(* Logix 5000 project; controller TBEN_Lx_8IOL_AOI_V0_2 vendor 1 type 14 code 176 rev 32.11; software revision 32.00; part 12 of 16 *)

           TBEN_L4_8IOL1:O.Data[69].10   // IO-Link Port 5 - Output data word 3 (INT bit10)
           TBEN_L4_8IOL1:O.Data[69].11   // IO-Link Port 5 - Output data word 3 (INT bit11)
           TBEN_L4_8IOL1:O.Data[69].12   // IO-Link Port 5 - Output data word 3 (INT bit12)
           TBEN_L4_8IOL1:O.Data[69].13   // IO-Link Port 5 - Output data word 3 (INT bit13)
           TBEN_L4_8IOL1:O.Data[69].14   // IO-Link Port 5 - Output data word 3 (INT bit14)
           TBEN_L4_8IOL1:O.Data[69].15   // IO-Link Port 5 - Output data word 3 (INT bit15)
           TBEN_L4_8IOL1:O.Data[69].2   // IO-Link Port 5 - Output data word 3 (INT bit2)
           TBEN_L4_8IOL1:O.Data[69].3   // IO-Link Port 5 - Output data word 3 (INT bit3)
           TBEN_L4_8IOL1:O.Data[69].4   // IO-Link Port 5 - Output data word 3 (INT bit4)
           TBEN_L4_8IOL1:O.Data[69].5   // IO-Link Port 5 - Output data word 3 (INT bit5)
           TBEN_L4_8IOL1:O.Data[69].6   // IO-Link Port 5 - Output data word 3 (INT bit6)
           TBEN_L4_8IOL1:O.Data[69].7   // IO-Link Port 5 - Output data word 3 (INT bit7)
           TBEN_L4_8IOL1:O.Data[69].8   // IO-Link Port 5 - Output data word 3 (INT bit8)
           TBEN_L4_8IOL1:O.Data[69].9   // IO-Link Port 5 - Output data word 3 (INT bit9)
           TBEN_L4_8IOL1:O.Data[6]   // IO-Link Port 1 - Output data word 4
           TBEN_L4_8IOL1:O.Data[6].0   // IO-Link Port 1 - Output data word 4 (INT bit0)
           TBEN_L4_8IOL1:O.Data[6].1   // IO-Link Port 1 - Output data word 4 (INT bit1)
           TBEN_L4_8IOL1:O.Data[6].10   // IO-Link Port 1 - Output data word 4 (INT bit10)
           TBEN_L4_8IOL1:O.Data[6].11   // IO-Link Port 1 - Output data word 4 (INT bit11)
           TBEN_L4_8IOL1:O.Data[6].12   // IO-Link Port 1 - Output data word 4 (INT bit12)
           TBEN_L4_8IOL1:O.Data[6].13   // IO-Link Port 1 - Output data word 4 (INT bit13)
           TBEN_L4_8IOL1:O.Data[6].14   // IO-Link Port 1 - Output data word 4 (INT bit14)
           TBEN_L4_8IOL1:O.Data[6].15   // IO-Link Port 1 - Output data word 4 (INT bit15)
           TBEN_L4_8IOL1:O.Data[6].2   // IO-Link Port 1 - Output data word 4 (INT bit2)
           TBEN_L4_8IOL1:O.Data[6].3   // IO-Link Port 1 - Output data word 4 (INT bit3)
           TBEN_L4_8IOL1:O.Data[6].4   // IO-Link Port 1 - Output data word 4 (INT bit4)
           TBEN_L4_8IOL1:O.Data[6].5   // IO-Link Port 1 - Output data word 4 (INT bit5)
           TBEN_L4_8IOL1:O.Data[6].6   // IO-Link Port 1 - Output data word 4 (INT bit6)
           TBEN_L4_8IOL1:O.Data[6].7   // IO-Link Port 1 - Output data word 4 (INT bit7)
           TBEN_L4_8IOL1:O.Data[6].8   // IO-Link Port 1 - Output data word 4 (INT bit8)
           TBEN_L4_8IOL1:O.Data[6].9   // IO-Link Port 1 - Output data word 4 (INT bit9)
           TBEN_L4_8IOL1:O.Data[70]   // IO-Link Port 5 - Output data word 4
           TBEN_L4_8IOL1:O.Data[70].0   // IO-Link Port 5 - Output data word 4 (INT bit0)
           TBEN_L4_8IOL1:O.Data[70].1   // IO-Link Port 5 - Output data word 4 (INT bit1)
           TBEN_L4_8IOL1:O.Data[70].10   // IO-Link Port 5 - Output data word 4 (INT bit10)
           TBEN_L4_8IOL1:O.Data[70].11   // IO-Link Port 5 - Output data word 4 (INT bit11)
           TBEN_L4_8IOL1:O.Data[70].12   // IO-Link Port 5 - Output data word 4 (INT bit12)
           TBEN_L4_8IOL1:O.Data[70].13   // IO-Link Port 5 - Output data word 4 (INT bit13)
           TBEN_L4_8IOL1:O.Data[70].14   // IO-Link Port 5 - Output data word 4 (INT bit14)
           TBEN_L4_8IOL1:O.Data[70].15   // IO-Link Port 5 - Output data word 4 (INT bit15)
           TBEN_L4_8IOL1:O.Data[70].2   // IO-Link Port 5 - Output data word 4 (INT bit2)
           TBEN_L4_8IOL1:O.Data[70].3   // IO-Link Port 5 - Output data word 4 (INT bit3)
           TBEN_L4_8IOL1:O.Data[70].4   // IO-Link Port 5 - Output data word 4 (INT bit4)
           TBEN_L4_8IOL1:O.Data[70].5   // IO-Link Port 5 - Output data word 4 (INT bit5)
           TBEN_L4_8IOL1:O.Data[70].6   // IO-Link Port 5 - Output data word 4 (INT bit6)
           TBEN_L4_8IOL1:O.Data[70].7   // IO-Link Port 5 - Output data word 4 (INT bit7)
           TBEN_L4_8IOL1:O.Data[70].8   // IO-Link Port 5 - Output data word 4 (INT bit8)
           TBEN_L4_8IOL1:O.Data[70].9   // IO-Link Port 5 - Output data word 4 (INT bit9)
           TBEN_L4_8IOL1:O.Data[71]   // IO-Link Port 5 - Output data word 5
           TBEN_L4_8IOL1:O.Data[71].0   // IO-Link Port 5 - Output data word 5 (INT bit0)
           TBEN_L4_8IOL1:O.Data[71].1   // IO-Link Port 5 - Output data word 5 (INT bit1)
           TBEN_L4_8IOL1:O.Data[71].10   // IO-Link Port 5 - Output data word 5 (INT bit10)
           TBEN_L4_8IOL1:O.Data[71].11   // IO-Link Port 5 - Output data word 5 (INT bit11)
           TBEN_L4_8IOL1:O.Data[71].12   // IO-Link Port 5 - Output data word 5 (INT bit12)
           TBEN_L4_8IOL1:O.Data[71].13   // IO-Link Port 5 - Output data word 5 (INT bit13)
           TBEN_L4_8IOL1:O.Data[71].14   // IO-Link Port 5 - Output data word 5 (INT bit14)
           TBEN_L4_8IOL1:O.Data[71].15   // IO-Link Port 5 - Output data word 5 (INT bit15)
           TBEN_L4_8IOL1:O.Data[71].2   // IO-Link Port 5 - Output data word 5 (INT bit2)
           TBEN_L4_8IOL1:O.Data[71].3   // IO-Link Port 5 - Output data word 5 (INT bit3)
           TBEN_L4_8IOL1:O.Data[71].4   // IO-Link Port 5 - Output data word 5 (INT bit4)
           TBEN_L4_8IOL1:O.Data[71].5   // IO-Link Port 5 - Output data word 5 (INT bit5)
           TBEN_L4_8IOL1:O.Data[71].6   // IO-Link Port 5 - Output data word 5 (INT bit6)
           TBEN_L4_8IOL1:O.Data[71].7   // IO-Link Port 5 - Output data word 5 (INT bit7)
           TBEN_L4_8IOL1:O.Data[71].8   // IO-Link Port 5 - Output data word 5 (INT bit8)
           TBEN_L4_8IOL1:O.Data[71].9   // IO-Link Port 5 - Output data word 5 (INT bit9)
           TBEN_L4_8IOL1:O.Data[72]   // IO-Link Port 5 - Output data word 6
           TBEN_L4_8IOL1:O.Data[72].0   // IO-Link Port 5 - Output data word 6 (INT bit0)
           TBEN_L4_8IOL1:O.Data[72].1   // IO-Link Port 5 - Output data word 6 (INT bit1)
           TBEN_L4_8IOL1:O.Data[72].10   // IO-Link Port 5 - Output data word 6 (INT bit10)
           TBEN_L4_8IOL1:O.Data[72].11   // IO-Link Port 5 - Output data word 6 (INT bit11)
           TBEN_L4_8IOL1:O.Data[72].12   // IO-Link Port 5 - Output data word 6 (INT bit12)
           TBEN_L4_8IOL1:O.Data[72].13   // IO-Link Port 5 - Output data word 6 (INT bit13)
           TBEN_L4_8IOL1:O.Data[72].14   // IO-Link Port 5 - Output data word 6 (INT bit14)
           TBEN_L4_8IOL1:O.Data[72].15   // IO-Link Port 5 - Output data word 6 (INT bit15)
           TBEN_L4_8IOL1:O.Data[72].2   // IO-Link Port 5 - Output data word 6 (INT bit2)
           TBEN_L4_8IOL1:O.Data[72].3   // IO-Link Port 5 - Output data word 6 (INT bit3)
           TBEN_L4_8IOL1:O.Data[72].4   // IO-Link Port 5 - Output data word 6 (INT bit4)
           TBEN_L4_8IOL1:O.Data[72].5   // IO-Link Port 5 - Output data word 6 (INT bit5)
           TBEN_L4_8IOL1:O.Data[72].6   // IO-Link Port 5 - Output data word 6 (INT bit6)
           TBEN_L4_8IOL1:O.Data[72].7   // IO-Link Port 5 - Output data word 6 (INT bit7)
           TBEN_L4_8IOL1:O.Data[72].8   // IO-Link Port 5 - Output data word 6 (INT bit8)
           TBEN_L4_8IOL1:O.Data[72].9   // IO-Link Port 5 - Output data word 6 (INT bit9)
           TBEN_L4_8IOL1:O.Data[73]   // IO-Link Port 5 - Output data word 7
           TBEN_L4_8IOL1:O.Data[73].0   // IO-Link Port 5 - Output data word 7 (INT bit0)
           TBEN_L4_8IOL1:O.Data[73].1   // IO-Link Port 5 - Output data word 7 (INT bit1)
           TBEN_L4_8IOL1:O.Data[73].10   // IO-Link Port 5 - Output data word 7 (INT bit10)
           TBEN_L4_8IOL1:O.Data[73].11   // IO-Link Port 5 - Output data word 7 (INT bit11)
           TBEN_L4_8IOL1:O.Data[73].12   // IO-Link Port 5 - Output data word 7 (INT bit12)
           TBEN_L4_8IOL1:O.Data[73].13   // IO-Link Port 5 - Output data word 7 (INT bit13)
           TBEN_L4_8IOL1:O.Data[73].14   // IO-Link Port 5 - Output data word 7 (INT bit14)
           TBEN_L4_8IOL1:O.Data[73].15   // IO-Link Port 5 - Output data word 7 (INT bit15)
           TBEN_L4_8IOL1:O.Data[73].2   // IO-Link Port 5 - Output data word 7 (INT bit2)
           TBEN_L4_8IOL1:O.Data[73].3   // IO-Link Port 5 - Output data word 7 (INT bit3)
           TBEN_L4_8IOL1:O.Data[73].4   // IO-Link Port 5 - Output data word 7 (INT bit4)
           TBEN_L4_8IOL1:O.Data[73].5   // IO-Link Port 5 - Output data word 7 (INT bit5)
           TBEN_L4_8IOL1:O.Data[73].6   // IO-Link Port 5 - Output data word 7 (INT bit6)
           TBEN_L4_8IOL1:O.Data[73].7   // IO-Link Port 5 - Output data word 7 (INT bit7)
           TBEN_L4_8IOL1:O.Data[73].8   // IO-Link Port 5 - Output data word 7 (INT bit8)
           TBEN_L4_8IOL1:O.Data[73].9   // IO-Link Port 5 - Output data word 7 (INT bit9)
           TBEN_L4_8IOL1:O.Data[74]   // IO-Link Port 5 - Output data word 8
           TBEN_L4_8IOL1:O.Data[74].0   // IO-Link Port 5 - Output data word 8 (INT bit0)
           TBEN_L4_8IOL1:O.Data[74].1   // IO-Link Port 5 - Output data word 8 (INT bit1)
           TBEN_L4_8IOL1:O.Data[74].10   // IO-Link Port 5 - Output data word 8 (INT bit10)
           TBEN_L4_8IOL1:O.Data[74].11   // IO-Link Port 5 - Output data word 8 (INT bit11)
           TBEN_L4_8IOL1:O.Data[74].12   // IO-Link Port 5 - Output data word 8 (INT bit12)
           TBEN_L4_8IOL1:O.Data[74].13   // IO-Link Port 5 - Output data word 8 (INT bit13)
           TBEN_L4_8IOL1:O.Data[74].14   // IO-Link Port 5 - Output data word 8 (INT bit14)
           TBEN_L4_8IOL1:O.Data[74].15   // IO-Link Port 5 - Output data word 8 (INT bit15)
           TBEN_L4_8IOL1:O.Data[74].2   // IO-Link Port 5 - Output data word 8 (INT bit2)
           TBEN_L4_8IOL1:O.Data[74].3   // IO-Link Port 5 - Output data word 8 (INT bit3)
           TBEN_L4_8IOL1:O.Data[74].4   // IO-Link Port 5 - Output data word 8 (INT bit4)
           TBEN_L4_8IOL1:O.Data[74].5   // IO-Link Port 5 - Output data word 8 (INT bit5)
           TBEN_L4_8IOL1:O.Data[74].6   // IO-Link Port 5 - Output data word 8 (INT bit6)
           TBEN_L4_8IOL1:O.Data[74].7   // IO-Link Port 5 - Output data word 8 (INT bit7)
           TBEN_L4_8IOL1:O.Data[74].8   // IO-Link Port 5 - Output data word 8 (INT bit8)
           TBEN_L4_8IOL1:O.Data[74].9   // IO-Link Port 5 - Output data word 8 (INT bit9)
           TBEN_L4_8IOL1:O.Data[75]   // IO-Link Port 5 - Output data word 9
           TBEN_L4_8IOL1:O.Data[75].0   // IO-Link Port 5 - Output data word 9 (INT bit0)
           TBEN_L4_8IOL1:O.Data[75].1   // IO-Link Port 5 - Output data word 9 (INT bit1)
           TBEN_L4_8IOL1:O.Data[75].10   // IO-Link Port 5 - Output data word 9 (INT bit10)
           TBEN_L4_8IOL1:O.Data[75].11   // IO-Link Port 5 - Output data word 9 (INT bit11)
           TBEN_L4_8IOL1:O.Data[75].12   // IO-Link Port 5 - Output data word 9 (INT bit12)
           TBEN_L4_8IOL1:O.Data[75].13   // IO-Link Port 5 - Output data word 9 (INT bit13)
           TBEN_L4_8IOL1:O.Data[75].14   // IO-Link Port 5 - Output data word 9 (INT bit14)
           TBEN_L4_8IOL1:O.Data[75].15   // IO-Link Port 5 - Output data word 9 (INT bit15)
           TBEN_L4_8IOL1:O.Data[75].2   // IO-Link Port 5 - Output data word 9 (INT bit2)
           TBEN_L4_8IOL1:O.Data[75].3   // IO-Link Port 5 - Output data word 9 (INT bit3)
           TBEN_L4_8IOL1:O.Data[75].4   // IO-Link Port 5 - Output data word 9 (INT bit4)
           TBEN_L4_8IOL1:O.Data[75].5   // IO-Link Port 5 - Output data word 9 (INT bit5)
           TBEN_L4_8IOL1:O.Data[75].6   // IO-Link Port 5 - Output data word 9 (INT bit6)
           TBEN_L4_8IOL1:O.Data[75].7   // IO-Link Port 5 - Output data word 9 (INT bit7)
           TBEN_L4_8IOL1:O.Data[75].8   // IO-Link Port 5 - Output data word 9 (INT bit8)
           TBEN_L4_8IOL1:O.Data[75].9   // IO-Link Port 5 - Output data word 9 (INT bit9)
           TBEN_L4_8IOL1:O.Data[76]   // IO-Link Port 5 - Output data word 10
           TBEN_L4_8IOL1:O.Data[76].0   // IO-Link Port 5 - Output data word 10 (INT bit0)
           TBEN_L4_8IOL1:O.Data[76].1   // IO-Link Port 5 - Output data word 10 (INT bit1)
           TBEN_L4_8IOL1:O.Data[76].10   // IO-Link Port 5 - Output data word 10 (INT bit10)
           TBEN_L4_8IOL1:O.Data[76].11   // IO-Link Port 5 - Output data word 10 (INT bit11)
           TBEN_L4_8IOL1:O.Data[76].12   // IO-Link Port 5 - Output data word 10 (INT bit12)
           TBEN_L4_8IOL1:O.Data[76].13   // IO-Link Port 5 - Output data word 10 (INT bit13)
           TBEN_L4_8IOL1:O.Data[76].14   // IO-Link Port 5 - Output data word 10 (INT bit14)
           TBEN_L4_8IOL1:O.Data[76].15   // IO-Link Port 5 - Output data word 10 (INT bit15)
           TBEN_L4_8IOL1:O.Data[76].2   // IO-Link Port 5 - Output data word 10 (INT bit2)
           TBEN_L4_8IOL1:O.Data[76].3   // IO-Link Port 5 - Output data word 10 (INT bit3)
           TBEN_L4_8IOL1:O.Data[76].4   // IO-Link Port 5 - Output data word 10 (INT bit4)
           TBEN_L4_8IOL1:O.Data[76].5   // IO-Link Port 5 - Output data word 10 (INT bit5)
           TBEN_L4_8IOL1:O.Data[76].6   // IO-Link Port 5 - Output data word 10 (INT bit6)
           TBEN_L4_8IOL1:O.Data[76].7   // IO-Link Port 5 - Output data word 10 (INT bit7)
           TBEN_L4_8IOL1:O.Data[76].8   // IO-Link Port 5 - Output data word 10 (INT bit8)
           TBEN_L4_8IOL1:O.Data[76].9   // IO-Link Port 5 - Output data word 10 (INT bit9)
           TBEN_L4_8IOL1:O.Data[77]   // IO-Link Port 5 - Output data word 11
           TBEN_L4_8IOL1:O.Data[77].0   // IO-Link Port 5 - Output data word 11 (INT bit0)
           TBEN_L4_8IOL1:O.Data[77].1   // IO-Link Port 5 - Output data word 11 (INT bit1)
           TBEN_L4_8IOL1:O.Data[77].10   // IO-Link Port 5 - Output data word 11 (INT bit10)
           TBEN_L4_8IOL1:O.Data[77].11   // IO-Link Port 5 - Output data word 11 (INT bit11)
           TBEN_L4_8IOL1:O.Data[77].12   // IO-Link Port 5 - Output data word 11 (INT bit12)
           TBEN_L4_8IOL1:O.Data[77].13   // IO-Link Port 5 - Output data word 11 (INT bit13)
           TBEN_L4_8IOL1:O.Data[77].14   // IO-Link Port 5 - Output data word 11 (INT bit14)
           TBEN_L4_8IOL1:O.Data[77].15   // IO-Link Port 5 - Output data word 11 (INT bit15)
           TBEN_L4_8IOL1:O.Data[77].2   // IO-Link Port 5 - Output data word 11 (INT bit2)
           TBEN_L4_8IOL1:O.Data[77].3   // IO-Link Port 5 - Output data word 11 (INT bit3)
           TBEN_L4_8IOL1:O.Data[77].4   // IO-Link Port 5 - Output data word 11 (INT bit4)
           TBEN_L4_8IOL1:O.Data[77].5   // IO-Link Port 5 - Output data word 11 (INT bit5)
           TBEN_L4_8IOL1:O.Data[77].6   // IO-Link Port 5 - Output data word 11 (INT bit6)
           TBEN_L4_8IOL1:O.Data[77].7   // IO-Link Port 5 - Output data word 11 (INT bit7)
           TBEN_L4_8IOL1:O.Data[77].8   // IO-Link Port 5 - Output data word 11 (INT bit8)
           TBEN_L4_8IOL1:O.Data[77].9   // IO-Link Port 5 - Output data word 11 (INT bit9)
           TBEN_L4_8IOL1:O.Data[78]   // IO-Link Port 5 - Output data word 12
           TBEN_L4_8IOL1:O.Data[78].0   // IO-Link Port 5 - Output data word 12 (INT bit0)
           TBEN_L4_8IOL1:O.Data[78].1   // IO-Link Port 5 - Output data word 12 (INT bit1)
           TBEN_L4_8IOL1:O.Data[78].10   // IO-Link Port 5 - Output data word 12 (INT bit10)
           TBEN_L4_8IOL1:O.Data[78].11   // IO-Link Port 5 - Output data word 12 (INT bit11)
           TBEN_L4_8IOL1:O.Data[78].12   // IO-Link Port 5 - Output data word 12 (INT bit12)
           TBEN_L4_8IOL1:O.Data[78].13   // IO-Link Port 5 - Output data word 12 (INT bit13)
           TBEN_L4_8IOL1:O.Data[78].14   // IO-Link Port 5 - Output data word 12 (INT bit14)
           TBEN_L4_8IOL1:O.Data[78].15   // IO-Link Port 5 - Output data word 12 (INT bit15)
           TBEN_L4_8IOL1:O.Data[78].2   // IO-Link Port 5 - Output data word 12 (INT bit2)
           TBEN_L4_8IOL1:O.Data[78].3   // IO-Link Port 5 - Output data word 12 (INT bit3)
           TBEN_L4_8IOL1:O.Data[78].4   // IO-Link Port 5 - Output data word 12 (INT bit4)
           TBEN_L4_8IOL1:O.Data[78].5   // IO-Link Port 5 - Output data word 12 (INT bit5)
           TBEN_L4_8IOL1:O.Data[78].6   // IO-Link Port 5 - Output data word 12 (INT bit6)
           TBEN_L4_8IOL1:O.Data[78].7   // IO-Link Port 5 - Output data word 12 (INT bit7)
           TBEN_L4_8IOL1:O.Data[78].8   // IO-Link Port 5 - Output data word 12 (INT bit8)
           TBEN_L4_8IOL1:O.Data[78].9   // IO-Link Port 5 - Output data word 12 (INT bit9)
           TBEN_L4_8IOL1:O.Data[79]   // IO-Link Port 5 - Output data word 13
           TBEN_L4_8IOL1:O.Data[79].0   // IO-Link Port 5 - Output data word 13 (INT bit0)
           TBEN_L4_8IOL1:O.Data[79].1   // IO-Link Port 5 - Output data word 13 (INT bit1)
           TBEN_L4_8IOL1:O.Data[79].10   // IO-Link Port 5 - Output data word 13 (INT bit10)
           TBEN_L4_8IOL1:O.Data[79].11   // IO-Link Port 5 - Output data word 13 (INT bit11)
           TBEN_L4_8IOL1:O.Data[79].12   // IO-Link Port 5 - Output data word 13 (INT bit12)
           TBEN_L4_8IOL1:O.Data[79].13   // IO-Link Port 5 - Output data word 13 (INT bit13)
           TBEN_L4_8IOL1:O.Data[79].14   // IO-Link Port 5 - Output data word 13 (INT bit14)
           TBEN_L4_8IOL1:O.Data[79].15   // IO-Link Port 5 - Output data word 13 (INT bit15)
           TBEN_L4_8IOL1:O.Data[79].2   // IO-Link Port 5 - Output data word 13 (INT bit2)
           TBEN_L4_8IOL1:O.Data[79].3   // IO-Link Port 5 - Output data word 13 (INT bit3)
           TBEN_L4_8IOL1:O.Data[79].4   // IO-Link Port 5 - Output data word 13 (INT bit4)
           TBEN_L4_8IOL1:O.Data[79].5   // IO-Link Port 5 - Output data word 13 (INT bit5)
           TBEN_L4_8IOL1:O.Data[79].6   // IO-Link Port 5 - Output data word 13 (INT bit6)
           TBEN_L4_8IOL1:O.Data[79].7   // IO-Link Port 5 - Output data word 13 (INT bit7)
           TBEN_L4_8IOL1:O.Data[79].8   // IO-Link Port 5 - Output data word 13 (INT bit8)
           TBEN_L4_8IOL1:O.Data[79].9   // IO-Link Port 5 - Output data word 13 (INT bit9)
           TBEN_L4_8IOL1:O.Data[7]   // IO-Link Port 1 - Output data word 5
           TBEN_L4_8IOL1:O.Data[7].0   // IO-Link Port 1 - Output data word 5 (INT bit0)
           TBEN_L4_8IOL1:O.Data[7].1   // IO-Link Port 1 - Output data word 5 (INT bit1)
           TBEN_L4_8IOL1:O.Data[7].10   // IO-Link Port 1 - Output data word 5 (INT bit10)
           TBEN_L4_8IOL1:O.Data[7].11   // IO-Link Port 1 - Output data word 5 (INT bit11)
           TBEN_L4_8IOL1:O.Data[7].12   // IO-Link Port 1 - Output data word 5 (INT bit12)
           TBEN_L4_8IOL1:O.Data[7].13   // IO-Link Port 1 - Output data word 5 (INT bit13)
           TBEN_L4_8IOL1:O.Data[7].14   // IO-Link Port 1 - Output data word 5 (INT bit14)
           TBEN_L4_8IOL1:O.Data[7].15   // IO-Link Port 1 - Output data word 5 (INT bit15)
           TBEN_L4_8IOL1:O.Data[7].2   // IO-Link Port 1 - Output data word 5 (INT bit2)
           TBEN_L4_8IOL1:O.Data[7].3   // IO-Link Port 1 - Output data word 5 (INT bit3)
           TBEN_L4_8IOL1:O.Data[7].4   // IO-Link Port 1 - Output data word 5 (INT bit4)
           TBEN_L4_8IOL1:O.Data[7].5   // IO-Link Port 1 - Output data word 5 (INT bit5)
           TBEN_L4_8IOL1:O.Data[7].6   // IO-Link Port 1 - Output data word 5 (INT bit6)
           TBEN_L4_8IOL1:O.Data[7].7   // IO-Link Port 1 - Output data word 5 (INT bit7)
           TBEN_L4_8IOL1:O.Data[7].8   // IO-Link Port 1 - Output data word 5 (INT bit8)
           TBEN_L4_8IOL1:O.Data[7].9   // IO-Link Port 1 - Output data word 5 (INT bit9)
           TBEN_L4_8IOL1:O.Data[80]   // IO-Link Port 5 - Output data word 14
           TBEN_L4_8IOL1:O.Data[80].0   // IO-Link Port 5 - Output data word 14 (INT bit0)
           TBEN_L4_8IOL1:O.Data[80].1   // IO-Link Port 5 - Output data word 14 (INT bit1)
           TBEN_L4_8IOL1:O.Data[80].10   // IO-Link Port 5 - Output data word 14 (INT bit10)
           TBEN_L4_8IOL1:O.Data[80].11   // IO-Link Port 5 - Output data word 14 (INT bit11)
           TBEN_L4_8IOL1:O.Data[80].12   // IO-Link Port 5 - Output data word 14 (INT bit12)
           TBEN_L4_8IOL1:O.Data[80].13   // IO-Link Port 5 - Output data word 14 (INT bit13)
           TBEN_L4_8IOL1:O.Data[80].14   // IO-Link Port 5 - Output data word 14 (INT bit14)
           TBEN_L4_8IOL1:O.Data[80].15   // IO-Link Port 5 - Output data word 14 (INT bit15)
           TBEN_L4_8IOL1:O.Data[80].2   // IO-Link Port 5 - Output data word 14 (INT bit2)
           TBEN_L4_8IOL1:O.Data[80].3   // IO-Link Port 5 - Output data word 14 (INT bit3)
           TBEN_L4_8IOL1:O.Data[80].4   // IO-Link Port 5 - Output data word 14 (INT bit4)
           TBEN_L4_8IOL1:O.Data[80].5   // IO-Link Port 5 - Output data word 14 (INT bit5)
           TBEN_L4_8IOL1:O.Data[80].6   // IO-Link Port 5 - Output data word 14 (INT bit6)
           TBEN_L4_8IOL1:O.Data[80].7   // IO-Link Port 5 - Output data word 14 (INT bit7)
           TBEN_L4_8IOL1:O.Data[80].8   // IO-Link Port 5 - Output data word 14 (INT bit8)
           TBEN_L4_8IOL1:O.Data[80].9   // IO-Link Port 5 - Output data word 14 (INT bit9)
           TBEN_L4_8IOL1:O.Data[81]   // IO-Link Port 5 - Output data word 15
           TBEN_L4_8IOL1:O.Data[81].0   // IO-Link Port 5 - Output data word 15 (INT bit0)
           TBEN_L4_8IOL1:O.Data[81].1   // IO-Link Port 5 - Output data word 15 (INT bit1)
           TBEN_L4_8IOL1:O.Data[81].10   // IO-Link Port 5 - Output data word 15 (INT bit10)
           TBEN_L4_8IOL1:O.Data[81].11   // IO-Link Port 5 - Output data word 15 (INT bit11)
           TBEN_L4_8IOL1:O.Data[81].12   // IO-Link Port 5 - Output data word 15 (INT bit12)
           TBEN_L4_8IOL1:O.Data[81].13   // IO-Link Port 5 - Output data word 15 (INT bit13)
           TBEN_L4_8IOL1:O.Data[81].14   // IO-Link Port 5 - Output data word 15 (INT bit14)
           TBEN_L4_8IOL1:O.Data[81].15   // IO-Link Port 5 - Output data word 15 (INT bit15)
           TBEN_L4_8IOL1:O.Data[81].2   // IO-Link Port 5 - Output data word 15 (INT bit2)
           TBEN_L4_8IOL1:O.Data[81].3   // IO-Link Port 5 - Output data word 15 (INT bit3)
           TBEN_L4_8IOL1:O.Data[81].4   // IO-Link Port 5 - Output data word 15 (INT bit4)
           TBEN_L4_8IOL1:O.Data[81].5   // IO-Link Port 5 - Output data word 15 (INT bit5)
           TBEN_L4_8IOL1:O.Data[81].6   // IO-Link Port 5 - Output data word 15 (INT bit6)
           TBEN_L4_8IOL1:O.Data[81].7   // IO-Link Port 5 - Output data word 15 (INT bit7)
           TBEN_L4_8IOL1:O.Data[81].8   // IO-Link Port 5 - Output data word 15 (INT bit8)
           TBEN_L4_8IOL1:O.Data[81].9   // IO-Link Port 5 - Output data word 15 (INT bit9)
           TBEN_L4_8IOL1:O.Data[82]   // IO-Link Port 6 - Output data word 0
           TBEN_L4_8IOL1:O.Data[82].0   // IO-Link Port 6 - Output data word 0 (INT bit0)
           TBEN_L4_8IOL1:O.Data[82].1   // IO-Link Port 6 - Output data word 0 (INT bit1)
           TBEN_L4_8IOL1:O.Data[82].10   // IO-Link Port 6 - Output data word 0 (INT bit10)
           TBEN_L4_8IOL1:O.Data[82].11   // IO-Link Port 6 - Output data word 0 (INT bit11)
           TBEN_L4_8IOL1:O.Data[82].12   // IO-Link Port 6 - Output data word 0 (INT bit12)
           TBEN_L4_8IOL1:O.Data[82].13   // IO-Link Port 6 - Output data word 0 (INT bit13)
           TBEN_L4_8IOL1:O.Data[82].14   // IO-Link Port 6 - Output data word 0 (INT bit14)
           TBEN_L4_8IOL1:O.Data[82].15   // IO-Link Port 6 - Output data word 0 (INT bit15)
           TBEN_L4_8IOL1:O.Data[82].2   // IO-Link Port 6 - Output data word 0 (INT bit2)
           TBEN_L4_8IOL1:O.Data[82].3   // IO-Link Port 6 - Output data word 0 (INT bit3)
           TBEN_L4_8IOL1:O.Data[82].4   // IO-Link Port 6 - Output data word 0 (INT bit4)
           TBEN_L4_8IOL1:O.Data[82].5   // IO-Link Port 6 - Output data word 0 (INT bit5)
           TBEN_L4_8IOL1:O.Data[82].6   // IO-Link Port 6 - Output data word 0 (INT bit6)
           TBEN_L4_8IOL1:O.Data[82].7   // IO-Link Port 6 - Output data word 0 (INT bit7)
           TBEN_L4_8IOL1:O.Data[82].8   // IO-Link Port 6 - Output data word 0 (INT bit8)
           TBEN_L4_8IOL1:O.Data[82].9   // IO-Link Port 6 - Output data word 0 (INT bit9)
           TBEN_L4_8IOL1:O.Data[83]   // IO-Link Port 6 - Output data word 1
           TBEN_L4_8IOL1:O.Data[83].0   // IO-Link Port 6 - Output data word 1 (INT bit0)
           TBEN_L4_8IOL1:O.Data[83].1   // IO-Link Port 6 - Output data word 1 (INT bit1)
           TBEN_L4_8IOL1:O.Data[83].10   // IO-Link Port 6 - Output data word 1 (INT bit10)
           TBEN_L4_8IOL1:O.Data[83].11   // IO-Link Port 6 - Output data word 1 (INT bit11)
           TBEN_L4_8IOL1:O.Data[83].12   // IO-Link Port 6 - Output data word 1 (INT bit12)
           TBEN_L4_8IOL1:O.Data[83].13   // IO-Link Port 6 - Output data word 1 (INT bit13)
           TBEN_L4_8IOL1:O.Data[83].14   // IO-Link Port 6 - Output data word 1 (INT bit14)
           TBEN_L4_8IOL1:O.Data[83].15   // IO-Link Port 6 - Output data word 1 (INT bit15)
           TBEN_L4_8IOL1:O.Data[83].2   // IO-Link Port 6 - Output data word 1 (INT bit2)
           TBEN_L4_8IOL1:O.Data[83].3   // IO-Link Port 6 - Output data word 1 (INT bit3)
           TBEN_L4_8IOL1:O.Data[83].4   // IO-Link Port 6 - Output data word 1 (INT bit4)
           TBEN_L4_8IOL1:O.Data[83].5   // IO-Link Port 6 - Output data word 1 (INT bit5)
           TBEN_L4_8IOL1:O.Data[83].6   // IO-Link Port 6 - Output data word 1 (INT bit6)
           TBEN_L4_8IOL1:O.Data[83].7   // IO-Link Port 6 - Output data word 1 (INT bit7)
           TBEN_L4_8IOL1:O.Data[83].8   // IO-Link Port 6 - Output data word 1 (INT bit8)
           TBEN_L4_8IOL1:O.Data[83].9   // IO-Link Port 6 - Output data word 1 (INT bit9)
           TBEN_L4_8IOL1:O.Data[84]   // IO-Link Port 6 - Output data word 2
           TBEN_L4_8IOL1:O.Data[84].0   // IO-Link Port 6 - Output data word 2 (INT bit0)
           TBEN_L4_8IOL1:O.Data[84].1   // IO-Link Port 6 - Output data word 2 (INT bit1)
           TBEN_L4_8IOL1:O.Data[84].10   // IO-Link Port 6 - Output data word 2 (INT bit10)
           TBEN_L4_8IOL1:O.Data[84].11   // IO-Link Port 6 - Output data word 2 (INT bit11)
           TBEN_L4_8IOL1:O.Data[84].12   // IO-Link Port 6 - Output data word 2 (INT bit12)
           TBEN_L4_8IOL1:O.Data[84].13   // IO-Link Port 6 - Output data word 2 (INT bit13)
           TBEN_L4_8IOL1:O.Data[84].14   // IO-Link Port 6 - Output data word 2 (INT bit14)
           TBEN_L4_8IOL1:O.Data[84].15   // IO-Link Port 6 - Output data word 2 (INT bit15)
           TBEN_L4_8IOL1:O.Data[84].2   // IO-Link Port 6 - Output data word 2 (INT bit2)
           TBEN_L4_8IOL1:O.Data[84].3   // IO-Link Port 6 - Output data word 2 (INT bit3)
           TBEN_L4_8IOL1:O.Data[84].4   // IO-Link Port 6 - Output data word 2 (INT bit4)
           TBEN_L4_8IOL1:O.Data[84].5   // IO-Link Port 6 - Output data word 2 (INT bit5)
           TBEN_L4_8IOL1:O.Data[84].6   // IO-Link Port 6 - Output data word 2 (INT bit6)
           TBEN_L4_8IOL1:O.Data[84].7   // IO-Link Port 6 - Output data word 2 (INT bit7)
           TBEN_L4_8IOL1:O.Data[84].8   // IO-Link Port 6 - Output data word 2 (INT bit8)
           TBEN_L4_8IOL1:O.Data[84].9   // IO-Link Port 6 - Output data word 2 (INT bit9)
           TBEN_L4_8IOL1:O.Data[85]   // IO-Link Port 6 - Output data word 3
           TBEN_L4_8IOL1:O.Data[85].0   // IO-Link Port 6 - Output data word 3 (INT bit0)
           TBEN_L4_8IOL1:O.Data[85].1   // IO-Link Port 6 - Output data word 3 (INT bit1)
           TBEN_L4_8IOL1:O.Data[85].10   // IO-Link Port 6 - Output data word 3 (INT bit10)
           TBEN_L4_8IOL1:O.Data[85].11   // IO-Link Port 6 - Output data word 3 (INT bit11)
           TBEN_L4_8IOL1:O.Data[85].12   // IO-Link Port 6 - Output data word 3 (INT bit12)
           TBEN_L4_8IOL1:O.Data[85].13   // IO-Link Port 6 - Output data word 3 (INT bit13)
           TBEN_L4_8IOL1:O.Data[85].14   // IO-Link Port 6 - Output data word 3 (INT bit14)
           TBEN_L4_8IOL1:O.Data[85].15   // IO-Link Port 6 - Output data word 3 (INT bit15)
           TBEN_L4_8IOL1:O.Data[85].2   // IO-Link Port 6 - Output data word 3 (INT bit2)
           TBEN_L4_8IOL1:O.Data[85].3   // IO-Link Port 6 - Output data word 3 (INT bit3)
           TBEN_L4_8IOL1:O.Data[85].4   // IO-Link Port 6 - Output data word 3 (INT bit4)
           TBEN_L4_8IOL1:O.Data[85].5   // IO-Link Port 6 - Output data word 3 (INT bit5)
           TBEN_L4_8IOL1:O.Data[85].6   // IO-Link Port 6 - Output data word 3 (INT bit6)
           TBEN_L4_8IOL1:O.Data[85].7   // IO-Link Port 6 - Output data word 3 (INT bit7)
           TBEN_L4_8IOL1:O.Data[85].8   // IO-Link Port 6 - Output data word 3 (INT bit8)
           TBEN_L4_8IOL1:O.Data[85].9   // IO-Link Port 6 - Output data word 3 (INT bit9)
           TBEN_L4_8IOL1:O.Data[86]   // IO-Link Port 6 - Output data word 4
           TBEN_L4_8IOL1:O.Data[86].0   // IO-Link Port 6 - Output data word 4 (INT bit0)
           TBEN_L4_8IOL1:O.Data[86].1   // IO-Link Port 6 - Output data word 4 (INT bit1)
           TBEN_L4_8IOL1:O.Data[86].10   // IO-Link Port 6 - Output data word 4 (INT bit10)
           TBEN_L4_8IOL1:O.Data[86].11   // IO-Link Port 6 - Output data word 4 (INT bit11)
           TBEN_L4_8IOL1:O.Data[86].12   // IO-Link Port 6 - Output data word 4 (INT bit12)
           TBEN_L4_8IOL1:O.Data[86].13   // IO-Link Port 6 - Output data word 4 (INT bit13)
           TBEN_L4_8IOL1:O.Data[86].14   // IO-Link Port 6 - Output data word 4 (INT bit14)
           TBEN_L4_8IOL1:O.Data[86].15   // IO-Link Port 6 - Output data word 4 (INT bit15)
           TBEN_L4_8IOL1:O.Data[86].2   // IO-Link Port 6 - Output data word 4 (INT bit2)
           TBEN_L4_8IOL1:O.Data[86].3   // IO-Link Port 6 - Output data word 4 (INT bit3)
           TBEN_L4_8IOL1:O.Data[86].4   // IO-Link Port 6 - Output data word 4 (INT bit4)
           TBEN_L4_8IOL1:O.Data[86].5   // IO-Link Port 6 - Output data word 4 (INT bit5)
           TBEN_L4_8IOL1:O.Data[86].6   // IO-Link Port 6 - Output data word 4 (INT bit6)
           TBEN_L4_8IOL1:O.Data[86].7   // IO-Link Port 6 - Output data word 4 (INT bit7)
           TBEN_L4_8IOL1:O.Data[86].8   // IO-Link Port 6 - Output data word 4 (INT bit8)
           TBEN_L4_8IOL1:O.Data[86].9   // IO-Link Port 6 - Output data word 4 (INT bit9)
           TBEN_L4_8IOL1:O.Data[87]   // IO-Link Port 6 - Output data word 5
           TBEN_L4_8IOL1:O.Data[87].0   // IO-Link Port 6 - Output data word 5 (INT bit0)
           TBEN_L4_8IOL1:O.Data[87].1   // IO-Link Port 6 - Output data word 5 (INT bit1)
           TBEN_L4_8IOL1:O.Data[87].10   // IO-Link Port 6 - Output data word 5 (INT bit10)
           TBEN_L4_8IOL1:O.Data[87].11   // IO-Link Port 6 - Output data word 5 (INT bit11)
           TBEN_L4_8IOL1:O.Data[87].12   // IO-Link Port 6 - Output data word 5 (INT bit12)
           TBEN_L4_8IOL1:O.Data[87].13   // IO-Link Port 6 - Output data word 5 (INT bit13)
           TBEN_L4_8IOL1:O.Data[87].14   // IO-Link Port 6 - Output data word 5 (INT bit14)
           TBEN_L4_8IOL1:O.Data[87].15   // IO-Link Port 6 - Output data word 5 (INT bit15)
           TBEN_L4_8IOL1:O.Data[87].2   // IO-Link Port 6 - Output data word 5 (INT bit2)
           TBEN_L4_8IOL1:O.Data[87].3   // IO-Link Port 6 - Output data word 5 (INT bit3)
           TBEN_L4_8IOL1:O.Data[87].4   // IO-Link Port 6 - Output data word 5 (INT bit4)
           TBEN_L4_8IOL1:O.Data[87].5   // IO-Link Port 6 - Output data word 5 (INT bit5)
           TBEN_L4_8IOL1:O.Data[87].6   // IO-Link Port 6 - Output data word 5 (INT bit6)
           TBEN_L4_8IOL1:O.Data[87].7   // IO-Link Port 6 - Output data word 5 (INT bit7)
           TBEN_L4_8IOL1:O.Data[87].8   // IO-Link Port 6 - Output data word 5 (INT bit8)
           TBEN_L4_8IOL1:O.Data[87].9   // IO-Link Port 6 - Output data word 5 (INT bit9)
           TBEN_L4_8IOL1:O.Data[88]   // IO-Link Port 6 - Output data word 6
           TBEN_L4_8IOL1:O.Data[88].0   // IO-Link Port 6 - Output data word 6 (INT bit0)
           TBEN_L4_8IOL1:O.Data[88].1   // IO-Link Port 6 - Output data word 6 (INT bit1)
           TBEN_L4_8IOL1:O.Data[88].10   // IO-Link Port 6 - Output data word 6 (INT bit10)
           TBEN_L4_8IOL1:O.Data[88].11   // IO-Link Port 6 - Output data word 6 (INT bit11)
           TBEN_L4_8IOL1:O.Data[88].12   // IO-Link Port 6 - Output data word 6 (INT bit12)
           TBEN_L4_8IOL1:O.Data[88].13   // IO-Link Port 6 - Output data word 6 (INT bit13)
           TBEN_L4_8IOL1:O.Data[88].14   // IO-Link Port 6 - Output data word 6 (INT bit14)
           TBEN_L4_8IOL1:O.Data[88].15   // IO-Link Port 6 - Output data word 6 (INT bit15)
           TBEN_L4_8IOL1:O.Data[88].2   // IO-Link Port 6 - Output data word 6 (INT bit2)
           TBEN_L4_8IOL1:O.Data[88].3   // IO-Link Port 6 - Output data word 6 (INT bit3)
           TBEN_L4_8IOL1:O.Data[88].4   // IO-Link Port 6 - Output data word 6 (INT bit4)
           TBEN_L4_8IOL1:O.Data[88].5   // IO-Link Port 6 - Output data word 6 (INT bit5)
           TBEN_L4_8IOL1:O.Data[88].6   // IO-Link Port 6 - Output data word 6 (INT bit6)
           TBEN_L4_8IOL1:O.Data[88].7   // IO-Link Port 6 - Output data word 6 (INT bit7)
           TBEN_L4_8IOL1:O.Data[88].8   // IO-Link Port 6 - Output data word 6 (INT bit8)
           TBEN_L4_8IOL1:O.Data[88].9   // IO-Link Port 6 - Output data word 6 (INT bit9)
           TBEN_L4_8IOL1:O.Data[89]   // IO-Link Port 6 - Output data word 7
           TBEN_L4_8IOL1:O.Data[89].0   // IO-Link Port 6 - Output data word 7 (INT bit0)
           TBEN_L4_8IOL1:O.Data[89].1   // IO-Link Port 6 - Output data word 7 (INT bit1)
           TBEN_L4_8IOL1:O.Data[89].10   // IO-Link Port 6 - Output data word 7 (INT bit10)
           TBEN_L4_8IOL1:O.Data[89].11   // IO-Link Port 6 - Output data word 7 (INT bit11)
           TBEN_L4_8IOL1:O.Data[89].12   // IO-Link Port 6 - Output data word 7 (INT bit12)
           TBEN_L4_8IOL1:O.Data[89].13   // IO-Link Port 6 - Output data word 7 (INT bit13)
           TBEN_L4_8IOL1:O.Data[89].14   // IO-Link Port 6 - Output data word 7 (INT bit14)
           TBEN_L4_8IOL1:O.Data[89].15   // IO-Link Port 6 - Output data word 7 (INT bit15)
           TBEN_L4_8IOL1:O.Data[89].2   // IO-Link Port 6 - Output data word 7 (INT bit2)
           TBEN_L4_8IOL1:O.Data[89].3   // IO-Link Port 6 - Output data word 7 (INT bit3)
           TBEN_L4_8IOL1:O.Data[89].4   // IO-Link Port 6 - Output data word 7 (INT bit4)
           TBEN_L4_8IOL1:O.Data[89].5   // IO-Link Port 6 - Output data word 7 (INT bit5)
           TBEN_L4_8IOL1:O.Data[89].6   // IO-Link Port 6 - Output data word 7 (INT bit6)
           TBEN_L4_8IOL1:O.Data[89].7   // IO-Link Port 6 - Output data word 7 (INT bit7)
           TBEN_L4_8IOL1:O.Data[89].8   // IO-Link Port 6 - Output data word 7 (INT bit8)
           TBEN_L4_8IOL1:O.Data[89].9   // IO-Link Port 6 - Output data word 7 (INT bit9)
           TBEN_L4_8IOL1:O.Data[8]   // IO-Link Port 1 - Output data word 6
           TBEN_L4_8IOL1:O.Data[8].0   // IO-Link Port 1 - Output data word 6 (INT bit0)
           TBEN_L4_8IOL1:O.Data[8].1   // IO-Link Port 1 - Output data word 6 (INT bit1)
           TBEN_L4_8IOL1:O.Data[8].10   // IO-Link Port 1 - Output data word 6 (INT bit10)
           TBEN_L4_8IOL1:O.Data[8].11   // IO-Link Port 1 - Output data word 6 (INT bit11)
           TBEN_L4_8IOL1:O.Data[8].12   // IO-Link Port 1 - Output data word 6 (INT bit12)
           TBEN_L4_8IOL1:O.Data[8].13   // IO-Link Port 1 - Output data word 6 (INT bit13)
           TBEN_L4_8IOL1:O.Data[8].14   // IO-Link Port 1 - Output data word 6 (INT bit14)
           TBEN_L4_8IOL1:O.Data[8].15   // IO-Link Port 1 - Output data word 6 (INT bit15)
           TBEN_L4_8IOL1:O.Data[8].2   // IO-Link Port 1 - Output data word 6 (INT bit2)
           TBEN_L4_8IOL1:O.Data[8].3   // IO-Link Port 1 - Output data word 6 (INT bit3)
           TBEN_L4_8IOL1:O.Data[8].4   // IO-Link Port 1 - Output data word 6 (INT bit4)
           TBEN_L4_8IOL1:O.Data[8].5   // IO-Link Port 1 - Output data word 6 (INT bit5)
           TBEN_L4_8IOL1:O.Data[8].6   // IO-Link Port 1 - Output data word 6 (INT bit6)
           TBEN_L4_8IOL1:O.Data[8].7   // IO-Link Port 1 - Output data word 6 (INT bit7)
           TBEN_L4_8IOL1:O.Data[8].8   // IO-Link Port 1 - Output data word 6 (INT bit8)
           TBEN_L4_8IOL1:O.Data[8].9   // IO-Link Port 1 - Output data word 6 (INT bit9)
           TBEN_L4_8IOL1:O.Data[90]   // IO-Link Port 6 - Output data word 8
           TBEN_L4_8IOL1:O.Data[90].0   // IO-Link Port 6 - Output data word 8 (INT bit0)
           TBEN_L4_8IOL1:O.Data[90].1   // IO-Link Port 6 - Output data word 8 (INT bit1)
           TBEN_L4_8IOL1:O.Data[90].10   // IO-Link Port 6 - Output data word 8 (INT bit10)
           TBEN_L4_8IOL1:O.Data[90].11   // IO-Link Port 6 - Output data word 8 (INT bit11)
           TBEN_L4_8IOL1:O.Data[90].12   // IO-Link Port 6 - Output data word 8 (INT bit12)
           TBEN_L4_8IOL1:O.Data[90].13   // IO-Link Port 6 - Output data word 8 (INT bit13)
           TBEN_L4_8IOL1:O.Data[90].14   // IO-Link Port 6 - Output data word 8 (INT bit14)
           TBEN_L4_8IOL1:O.Data[90].15   // IO-Link Port 6 - Output data word 8 (INT bit15)
           TBEN_L4_8IOL1:O.Data[90].2   // IO-Link Port 6 - Output data word 8 (INT bit2)
           TBEN_L4_8IOL1:O.Data[90].3   // IO-Link Port 6 - Output data word 8 (INT bit3)
           TBEN_L4_8IOL1:O.Data[90].4   // IO-Link Port 6 - Output data word 8 (INT bit4)
           TBEN_L4_8IOL1:O.Data[90].5   // IO-Link Port 6 - Output data word 8 (INT bit5)
           TBEN_L4_8IOL1:O.Data[90].6   // IO-Link Port 6 - Output data word 8 (INT bit6)
           TBEN_L4_8IOL1:O.Data[90].7   // IO-Link Port 6 - Output data word 8 (INT bit7)
           TBEN_L4_8IOL1:O.Data[90].8   // IO-Link Port 6 - Output data word 8 (INT bit8)
           TBEN_L4_8IOL1:O.Data[90].9   // IO-Link Port 6 - Output data word 8 (INT bit9)
           TBEN_L4_8IOL1:O.Data[91]   // IO-Link Port 6 - Output data word 9
           TBEN_L4_8IOL1:O.Data[91].0   // IO-Link Port 6 - Output data word 9 (INT bit0)
           TBEN_L4_8IOL1:O.Data[91].1   // IO-Link Port 6 - Output data word 9 (INT bit1)
           TBEN_L4_8IOL1:O.Data[91].10   // IO-Link Port 6 - Output data word 9 (INT bit10)
           TBEN_L4_8IOL1:O.Data[91].11   // IO-Link Port 6 - Output data word 9 (INT bit11)
           TBEN_L4_8IOL1:O.Data[91].12   // IO-Link Port 6 - Output data word 9 (INT bit12)
           TBEN_L4_8IOL1:O.Data[91].13   // IO-Link Port 6 - Output data word 9 (INT bit13)
           TBEN_L4_8IOL1:O.Data[91].14   // IO-Link Port 6 - Output data word 9 (INT bit14)
           TBEN_L4_8IOL1:O.Data[91].15   // IO-Link Port 6 - Output data word 9 (INT bit15)
           TBEN_L4_8IOL1:O.Data[91].2   // IO-Link Port 6 - Output data word 9 (INT bit2)
           TBEN_L4_8IOL1:O.Data[91].3   // IO-Link Port 6 - Output data word 9 (INT bit3)
           TBEN_L4_8IOL1:O.Data[91].4   // IO-Link Port 6 - Output data word 9 (INT bit4)
           TBEN_L4_8IOL1:O.Data[91].5   // IO-Link Port 6 - Output data word 9 (INT bit5)
           TBEN_L4_8IOL1:O.Data[91].6   // IO-Link Port 6 - Output data word 9 (INT bit6)
           TBEN_L4_8IOL1:O.Data[91].7   // IO-Link Port 6 - Output data word 9 (INT bit7)
           TBEN_L4_8IOL1:O.Data[91].8   // IO-Link Port 6 - Output data word 9 (INT bit8)
           TBEN_L4_8IOL1:O.Data[91].9   // IO-Link Port 6 - Output data word 9 (INT bit9)
           TBEN_L4_8IOL1:O.Data[92]   // IO-Link Port 6 - Output data word 10
           TBEN_L4_8IOL1:O.Data[92].0   // IO-Link Port 6 - Output data word 10 (INT bit0)
           TBEN_L4_8IOL1:O.Data[92].1   // IO-Link Port 6 - Output data word 10 (INT bit1)
           TBEN_L4_8IOL1:O.Data[92].10   // IO-Link Port 6 - Output data word 10 (INT bit10)
           TBEN_L4_8IOL1:O.Data[92].11   // IO-Link Port 6 - Output data word 10 (INT bit11)
           TBEN_L4_8IOL1:O.Data[92].12   // IO-Link Port 6 - Output data word 10 (INT bit12)
           TBEN_L4_8IOL1:O.Data[92].13   // IO-Link Port 6 - Output data word 10 (INT bit13)
           TBEN_L4_8IOL1:O.Data[92].14   // IO-Link Port 6 - Output data word 10 (INT bit14)
           TBEN_L4_8IOL1:O.Data[92].15   // IO-Link Port 6 - Output data word 10 (INT bit15)
           TBEN_L4_8IOL1:O.Data[92].2   // IO-Link Port 6 - Output data word 10 (INT bit2)
           TBEN_L4_8IOL1:O.Data[92].3   // IO-Link Port 6 - Output data word 10 (INT bit3)
           TBEN_L4_8IOL1:O.Data[92].4   // IO-Link Port 6 - Output data word 10 (INT bit4)
           TBEN_L4_8IOL1:O.Data[92].5   // IO-Link Port 6 - Output data word 10 (INT bit5)
           TBEN_L4_8IOL1:O.Data[92].6   // IO-Link Port 6 - Output data word 10 (INT bit6)
           TBEN_L4_8IOL1:O.Data[92].7   // IO-Link Port 6 - Output data word 10 (INT bit7)
           TBEN_L4_8IOL1:O.Data[92].8   // IO-Link Port 6 - Output data word 10 (INT bit8)
           TBEN_L4_8IOL1:O.Data[92].9   // IO-Link Port 6 - Output data word 10 (INT bit9)
           TBEN_L4_8IOL1:O.Data[93]   // IO-Link Port 6 - Output data word 11
           TBEN_L4_8IOL1:O.Data[93].0   // IO-Link Port 6 - Output data word 11 (INT bit0)
           TBEN_L4_8IOL1:O.Data[93].1   // IO-Link Port 6 - Output data word 11 (INT bit1)
           TBEN_L4_8IOL1:O.Data[93].10   // IO-Link Port 6 - Output data word 11 (INT bit10)
           TBEN_L4_8IOL1:O.Data[93].11   // IO-Link Port 6 - Output data word 11 (INT bit11)
           TBEN_L4_8IOL1:O.Data[93].12   // IO-Link Port 6 - Output data word 11 (INT bit12)
           TBEN_L4_8IOL1:O.Data[93].13   // IO-Link Port 6 - Output data word 11 (INT bit13)
           TBEN_L4_8IOL1:O.Data[93].14   // IO-Link Port 6 - Output data word 11 (INT bit14)
           TBEN_L4_8IOL1:O.Data[93].15   // IO-Link Port 6 - Output data word 11 (INT bit15)
           TBEN_L4_8IOL1:O.Data[93].2   // IO-Link Port 6 - Output data word 11 (INT bit2)
           TBEN_L4_8IOL1:O.Data[93].3   // IO-Link Port 6 - Output data word 11 (INT bit3)
           TBEN_L4_8IOL1:O.Data[93].4   // IO-Link Port 6 - Output data word 11 (INT bit4)
           TBEN_L4_8IOL1:O.Data[93].5   // IO-Link Port 6 - Output data word 11 (INT bit5)
           TBEN_L4_8IOL1:O.Data[93].6   // IO-Link Port 6 - Output data word 11 (INT bit6)
           TBEN_L4_8IOL1:O.Data[93].7   // IO-Link Port 6 - Output data word 11 (INT bit7)
           TBEN_L4_8IOL1:O.Data[93].8   // IO-Link Port 6 - Output data word 11 (INT bit8)
           TBEN_L4_8IOL1:O.Data[93].9   // IO-Link Port 6 - Output data word 11 (INT bit9)
           TBEN_L4_8IOL1:O.Data[94]   // IO-Link Port 6 - Output data word 12
           TBEN_L4_8IOL1:O.Data[94].0   // IO-Link Port 6 - Output data word 12 (INT bit0)
           TBEN_L4_8IOL1:O.Data[94].1   // IO-Link Port 6 - Output data word 12 (INT bit1)
           TBEN_L4_8IOL1:O.Data[94].10   // IO-Link Port 6 - Output data word 12 (INT bit10)
           TBEN_L4_8IOL1:O.Data[94].11   // IO-Link Port 6 - Output data word 12 (INT bit11)
           TBEN_L4_8IOL1:O.Data[94].12   // IO-Link Port 6 - Output data word 12 (INT bit12)
           TBEN_L4_8IOL1:O.Data[94].13   // IO-Link Port 6 - Output data word 12 (INT bit13)
           TBEN_L4_8IOL1:O.Data[94].14   // IO-Link Port 6 - Output data word 12 (INT bit14)
           TBEN_L4_8IOL1:O.Data[94].15   // IO-Link Port 6 - Output data word 12 (INT bit15)
           TBEN_L4_8IOL1:O.Data[94].2   // IO-Link Port 6 - Output data word 12 (INT bit2)
           TBEN_L4_8IOL1:O.Data[94].3   // IO-Link Port 6 - Output data word 12 (INT bit3)
           TBEN_L4_8IOL1:O.Data[94].4   // IO-Link Port 6 - Output data word 12 (INT bit4)
           TBEN_L4_8IOL1:O.Data[94].5   // IO-Link Port 6 - Output data word 12 (INT bit5)
           TBEN_L4_8IOL1:O.Data[94].6   // IO-Link Port 6 - Output data word 12 (INT bit6)
           TBEN_L4_8IOL1:O.Data[94].7   // IO-Link Port 6 - Output data word 12 (INT bit7)
           TBEN_L4_8IOL1:O.Data[94].8   // IO-Link Port 6 - Output data word 12 (INT bit8)
           TBEN_L4_8IOL1:O.Data[94].9   // IO-Link Port 6 - Output data word 12 (INT bit9)
           TBEN_L4_8IOL1:O.Data[95]   // IO-Link Port 6 - Output data word 13
           TBEN_L4_8IOL1:O.Data[95].0   // IO-Link Port 6 - Output data word 13 (INT bit0)
           TBEN_L4_8IOL1:O.Data[95].1   // IO-Link Port 6 - Output data word 13 (INT bit1)
           TBEN_L4_8IOL1:O.Data[95].10   // IO-Link Port 6 - Output data word 13 (INT bit10)
           TBEN_L4_8IOL1:O.Data[95].11   // IO-Link Port 6 - Output data word 13 (INT bit11)
           TBEN_L4_8IOL1:O.Data[95].12   // IO-Link Port 6 - Output data word 13 (INT bit12)
           TBEN_L4_8IOL1:O.Data[95].13   // IO-Link Port 6 - Output data word 13 (INT bit13)
           TBEN_L4_8IOL1:O.Data[95].14   // IO-Link Port 6 - Output data word 13 (INT bit14)
           TBEN_L4_8IOL1:O.Data[95].15   // IO-Link Port 6 - Output data word 13 (INT bit15)
           TBEN_L4_8IOL1:O.Data[95].2   // IO-Link Port 6 - Output data word 13 (INT bit2)
           TBEN_L4_8IOL1:O.Data[95].3   // IO-Link Port 6 - Output data word 13 (INT bit3)
           TBEN_L4_8IOL1:O.Data[95].4   // IO-Link Port 6 - Output data word 13 (INT bit4)
           TBEN_L4_8IOL1:O.Data[95].5   // IO-Link Port 6 - Output data word 13 (INT bit5)
           TBEN_L4_8IOL1:O.Data[95].6   // IO-Link Port 6 - Output data word 13 (INT bit6)
           TBEN_L4_8IOL1:O.Data[95].7   // IO-Link Port 6 - Output data word 13 (INT bit7)
           TBEN_L4_8IOL1:O.Data[95].8   // IO-Link Port 6 - Output data word 13 (INT bit8)
           TBEN_L4_8IOL1:O.Data[95].9   // IO-Link Port 6 - Output data word 13 (INT bit9)
           TBEN_L4_8IOL1:O.Data[96]   // IO-Link Port 6 - Output data word 14
           TBEN_L4_8IOL1:O.Data[96].0   // IO-Link Port 6 - Output data word 14 (INT bit0)
           TBEN_L4_8IOL1:O.Data[96].1   // IO-Link Port 6 - Output data word 14 (INT bit1)
           TBEN_L4_8IOL1:O.Data[96].10   // IO-Link Port 6 - Output data word 14 (INT bit10)
           TBEN_L4_8IOL1:O.Data[96].11   // IO-Link Port 6 - Output data word 14 (INT bit11)
           TBEN_L4_8IOL1:O.Data[96].12   // IO-Link Port 6 - Output data word 14 (INT bit12)
           TBEN_L4_8IOL1:O.Data[96].13   // IO-Link Port 6 - Output data word 14 (INT bit13)
           TBEN_L4_8IOL1:O.Data[96].14   // IO-Link Port 6 - Output data word 14 (INT bit14)
           TBEN_L4_8IOL1:O.Data[96].15   // IO-Link Port 6 - Output data word 14 (INT bit15)
           TBEN_L4_8IOL1:O.Data[96].2   // IO-Link Port 6 - Output data word 14 (INT bit2)
           TBEN_L4_8IOL1:O.Data[96].3   // IO-Link Port 6 - Output data word 14 (INT bit3)
           TBEN_L4_8IOL1:O.Data[96].4   // IO-Link Port 6 - Output data word 14 (INT bit4)
           TBEN_L4_8IOL1:O.Data[96].5   // IO-Link Port 6 - Output data word 14 (INT bit5)
           TBEN_L4_8IOL1:O.Data[96].6   // IO-Link Port 6 - Output data word 14 (INT bit6)
           TBEN_L4_8IOL1:O.Data[96].7   // IO-Link Port 6 - Output data word 14 (INT bit7)
           TBEN_L4_8IOL1:O.Data[96].8   // IO-Link Port 6 - Output data word 14 (INT bit8)
           TBEN_L4_8IOL1:O.Data[96].9   // IO-Link Port 6 - Output data word 14 (INT bit9)
           TBEN_L4_8IOL1:O.Data[97]   // IO-Link Port 6 - Output data word 15
           TBEN_L4_8IOL1:O.Data[97].0   // IO-Link Port 6 - Output data word 15 (INT bit0)
           TBEN_L4_8IOL1:O.Data[97].1   // IO-Link Port 6 - Output data word 15 (INT bit1)
           TBEN_L4_8IOL1:O.Data[97].10   // IO-Link Port 6 - Output data word 15 (INT bit10)
           TBEN_L4_8IOL1:O.Data[97].11   // IO-Link Port 6 - Output data word 15 (INT bit11)
           TBEN_L4_8IOL1:O.Data[97].12   // IO-Link Port 6 - Output data word 15 (INT bit12)
           TBEN_L4_8IOL1:O.Data[97].13   // IO-Link Port 6 - Output data word 15 (INT bit13)
           TBEN_L4_8IOL1:O.Data[97].14   // IO-Link Port 6 - Output data word 15 (INT bit14)
           TBEN_L4_8IOL1:O.Data[97].15   // IO-Link Port 6 - Output data word 15 (INT bit15)
           TBEN_L4_8IOL1:O.Data[97].2   // IO-Link Port 6 - Output data word 15 (INT bit2)
           TBEN_L4_8IOL1:O.Data[97].3   // IO-Link Port 6 - Output data word 15 (INT bit3)
           TBEN_L4_8IOL1:O.Data[97].4   // IO-Link Port 6 - Output data word 15 (INT bit4)
           TBEN_L4_8IOL1:O.Data[97].5   // IO-Link Port 6 - Output data word 15 (INT bit5)
           TBEN_L4_8IOL1:O.Data[97].6   // IO-Link Port 6 - Output data word 15 (INT bit6)
           TBEN_L4_8IOL1:O.Data[97].7   // IO-Link Port 6 - Output data word 15 (INT bit7)
           TBEN_L4_8IOL1:O.Data[97].8   // IO-Link Port 6 - Output data word 15 (INT bit8)
           TBEN_L4_8IOL1:O.Data[97].9   // IO-Link Port 6 - Output data word 15 (INT bit9)
           TBEN_L4_8IOL1:O.Data[98]   // IO-Link Port 7 - Output data word 0
           TBEN_L4_8IOL1:O.Data[98].0   // IO-Link Port 7 - Output data word 0 (INT bit0)
           TBEN_L4_8IOL1:O.Data[98].1   // IO-Link Port 7 - Output data word 0 (INT bit1)
           TBEN_L4_8IOL1:O.Data[98].10   // IO-Link Port 7 - Output data word 0 (INT bit10)
           TBEN_L4_8IOL1:O.Data[98].11   // IO-Link Port 7 - Output data word 0 (INT bit11)
           TBEN_L4_8IOL1:O.Data[98].12   // IO-Link Port 7 - Output data word 0 (INT bit12)
           TBEN_L4_8IOL1:O.Data[98].13   // IO-Link Port 7 - Output data word 0 (INT bit13)
           TBEN_L4_8IOL1:O.Data[98].14   // IO-Link Port 7 - Output data word 0 (INT bit14)
           TBEN_L4_8IOL1:O.Data[98].15   // IO-Link Port 7 - Output data word 0 (INT bit15)
           TBEN_L4_8IOL1:O.Data[98].2   // IO-Link Port 7 - Output data word 0 (INT bit2)
           TBEN_L4_8IOL1:O.Data[98].3   // IO-Link Port 7 - Output data word 0 (INT bit3)
           TBEN_L4_8IOL1:O.Data[98].4   // IO-Link Port 7 - Output data word 0 (INT bit4)
           TBEN_L4_8IOL1:O.Data[98].5   // IO-Link Port 7 - Output data word 0 (INT bit5)
           TBEN_L4_8IOL1:O.Data[98].6   // IO-Link Port 7 - Output data word 0 (INT bit6)
           TBEN_L4_8IOL1:O.Data[98].7   // IO-Link Port 7 - Output data word 0 (INT bit7)
           TBEN_L4_8IOL1:O.Data[98].8   // IO-Link Port 7 - Output data word 0 (INT bit8)
           TBEN_L4_8IOL1:O.Data[98].9   // IO-Link Port 7 - Output data word 0 (INT bit9)
           TBEN_L4_8IOL1:O.Data[99]   // IO-Link Port 7 - Output data word 1
           TBEN_L4_8IOL1:O.Data[99].0   // IO-Link Port 7 - Output data word 1 (INT bit0)
           TBEN_L4_8IOL1:O.Data[99].1   // IO-Link Port 7 - Output data word 1 (INT bit1)
           TBEN_L4_8IOL1:O.Data[99].10   // IO-Link Port 7 - Output data word 1 (INT bit10)
           TBEN_L4_8IOL1:O.Data[99].11   // IO-Link Port 7 - Output data word 1 (INT bit11)
           TBEN_L4_8IOL1:O.Data[99].12   // IO-Link Port 7 - Output data word 1 (INT bit12)
           TBEN_L4_8IOL1:O.Data[99].13   // IO-Link Port 7 - Output data word 1 (INT bit13)
           TBEN_L4_8IOL1:O.Data[99].14   // IO-Link Port 7 - Output data word 1 (INT bit14)
           TBEN_L4_8IOL1:O.Data[99].15   // IO-Link Port 7 - Output data word 1 (INT bit15)
           TBEN_L4_8IOL1:O.Data[99].2   // IO-Link Port 7 - Output data word 1 (INT bit2)
           TBEN_L4_8IOL1:O.Data[99].3   // IO-Link Port 7 - Output data word 1 (INT bit3)
           TBEN_L4_8IOL1:O.Data[99].4   // IO-Link Port 7 - Output data word 1 (INT bit4)
           TBEN_L4_8IOL1:O.Data[99].5   // IO-Link Port 7 - Output data word 1 (INT bit5)
           TBEN_L4_8IOL1:O.Data[99].6   // IO-Link Port 7 - Output data word 1 (INT bit6)
           TBEN_L4_8IOL1:O.Data[99].7   // IO-Link Port 7 - Output data word 1 (INT bit7)
           TBEN_L4_8IOL1:O.Data[99].8   // IO-Link Port 7 - Output data word 1 (INT bit8)
           TBEN_L4_8IOL1:O.Data[99].9   // IO-Link Port 7 - Output data word 1 (INT bit9)
           TBEN_L4_8IOL1:O.Data[9]   // IO-Link Port 1 - Output data word 7
           TBEN_L4_8IOL1:O.Data[9].0   // IO-Link Port 1 - Output data word 7 (INT bit0)
           TBEN_L4_8IOL1:O.Data[9].1   // IO-Link Port 1 - Output data word 7 (INT bit1)
           TBEN_L4_8IOL1:O.Data[9].10   // IO-Link Port 1 - Output data word 7 (INT bit10)
           TBEN_L4_8IOL1:O.Data[9].11   // IO-Link Port 1 - Output data word 7 (INT bit11)
           TBEN_L4_8IOL1:O.Data[9].12   // IO-Link Port 1 - Output data word 7 (INT bit12)
           TBEN_L4_8IOL1:O.Data[9].13   // IO-Link Port 1 - Output data word 7 (INT bit13)
           TBEN_L4_8IOL1:O.Data[9].14   // IO-Link Port 1 - Output data word 7 (INT bit14)
           TBEN_L4_8IOL1:O.Data[9].15   // IO-Link Port 1 - Output data word 7 (INT bit15)
           TBEN_L4_8IOL1:O.Data[9].2   // IO-Link Port 1 - Output data word 7 (INT bit2)
           TBEN_L4_8IOL1:O.Data[9].3   // IO-Link Port 1 - Output data word 7 (INT bit3)
           TBEN_L4_8IOL1:O.Data[9].4   // IO-Link Port 1 - Output data word 7 (INT bit4)
           TBEN_L4_8IOL1:O.Data[9].5   // IO-Link Port 1 - Output data word 7 (INT bit5)
           TBEN_L4_8IOL1:O.Data[9].6   // IO-Link Port 1 - Output data word 7 (INT bit6)
           TBEN_L4_8IOL1:O.Data[9].7   // IO-Link Port 1 - Output data word 7 (INT bit7)
           TBEN_L4_8IOL1:O.Data[9].8   // IO-Link Port 1 - Output data word 7 (INT bit8)
           TBEN_L4_8IOL1:O.Data[9].9   // IO-Link Port 1 - Output data word 7 (INT bit9)
END_MODULES

TYPE Generic_131_Words :
STRUCT
   Data : INT[131];
END_STRUCT
END_TYPE

TYPE Generic_160_SINT :
STRUCT
   DATA : SINT[160];
END_STRUCT
END_TYPE

TYPE Generic_16_Words :
STRUCT
   Data : INT[16];
END_STRUCT
END_TYPE

TYPE Generic_173_Words :
STRUCT
   Data : INT[173];
END_STRUCT
END_TYPE

TYPE Generic_5_Words :
STRUCT
   Data : INT[5];
END_STRUCT
END_TYPE

TYPE IOLRequest :
STRUCT
   Enable_Multiple_Nodes : BOOL;   // Set to 1 to enable multiple nodes
   ApplicationPath : STRING;   // Set Path for following IOL Instructions
   Read : BOOL;   // For internal use to integrate IOLRead and IOWrite with IOLService
   Write : BOOL;   // For internal use to integrate IOLRead and IOWrite with IOLService
   Reset : BOOL;   // For internal use to integrate IOLRead and IOWrite with IOLService
   Done : BOOL;   // For internal use to integrate IOLRead and IOWrite with IOLService
   Error : BOOL;   // For internal use to integrate IOLRead and IOWrite with IOLService
   Slot : INT;   // For internal use to integrate IOLRead and IOWrite with IOLService
   Port : INT;   // For internal use to integrate IOLRead and IOWrite with IOLService
   Index : INT;   // For internal use to integrate IOLRead and IOWrite with IOLService
   SubIndex : INT;   // For internal use to integrate IOLRead and IOWrite with IOLService
   Length : INT;   // For internal use to integrate IOLRead and IOWrite with IOLService
   Handle : INT;   // For internal use to integrate IOLRead and IOWrite with IOLService
   Status : INT;   // For internal use to integrate IOLRead and IOWrite with IOLService
   NextHandle : INT;   // For internal use to integrate IOLRead and IOWrite with IOLService
   ReceiveData : SINT[145];   // For internal use to integrate IOLRead and IOWrite with IOLService
   SendData : SINT[145];   // For internal use to integrate IOLRead and IOWrite with IOLService
   WriteData : DINT;   // For internal use to integrate IOLRead and IOWrite with IOLService
   ActivePath : STRING;   // For internal use to integrate IOLRead and IOWrite with IOLService
END_STRUCT
END_TYPE

TYPE Turck_IOLink_Common_Data :
STRUCT
   Read : BOOL;   // For internal use to integrate IOLRead and IOWrite with IOLService
   Write : BOOL;   // For internal use to integrate IOLRead and IOWrite with IOLService
   Reset : BOOL;   // For internal use to integrate IOLRead and IOWrite with IOLService
   Done : BOOL;   // For internal use to integrate IOLRead and IOWrite with IOLService
   Error : BOOL;   // For internal use to integrate IOLRead and IOWrite with IOLService
   Port_in_Use : SINT;   // Each bit is set to show that a port is in use. If it's not in use the port diagnostics will be disabled so IO-Link can still be used but won't throw a red light if no device plugged
   Port : INT;   // For internal use to integrate IOLRead and IOWrite with IOLService
   Index : INT;   // For internal use to integrate IOLRead and IOWrite with IOLService
   SubIndex : INT;   // For internal use to integrate IOLRead and IOWrite with IOLService
   Length : INT;   // For internal use to integrate IOLRead and IOWrite with IOLService
   TicketNum : INT;   // For internal use to integrate IOLRead and IOWrite with IOLService
   Status : INT;   // For internal use to integrate IOLRead and IOWrite with IOLService
   NextTicketNum : INT;   // For internal use to integrate IOLRead and IOWrite with IOLService
   ReceiveData : SINT[255];   // For internal use to integrate IOLRead and IOWrite with IOLService
   SendData : SINT[145];   // For internal use to integrate IOLRead and IOWrite with IOLService
   Vendor_IDs : INT[8];
   Device_IDs : DINT[8];
   WriteData : DINT;
   Process_Input_Data : Generic_16_Words[8];
   Process_Output_Data : Generic_16_Words[8];
END_STRUCT
END_TYPE

TYPE Universal_IOLink_Info :
STRUCT
   Vendor_Name : STRING;   // Index 16
   Vendor_Text : STRING;   // Index 17
   Product_Name : STRING;   // Index 18
   Product_ID : STRING;   // Index 19
   Product_Text : STRING;   // Index 20
   Serial_Number : STRING;   // Index 21
   Hardware_Revision : STRING;   // Index 22
   Firmware_Revision : STRING;   // Index 23
   Application_Specific_Tag : STRING;   // Index 24
   Function_Tag : STRING;   // Index 25
   Location_Tag : STRING;   // Index 26
   Application_Specific_Tag_Requested : STRING;
END_STRUCT
END_TYPE

ADD_ON_INSTRUCTION IOL_ReadData   (* revision 2.5 Support TBIP, ExecutePrescan, ExecuteEnableInFalse *)
// Revision note:
// V1_0 Initial Release
// V1_1 Automatic data precision detection
// V1_2 Added multiple EIP node support
// V2_5 Support TBIP
// Help:
// IOL_ReadData - used with Turck BL20, BL67, BLC and TBEN IOLink masters to read numeric data from IOLink devices.  Use in conjuction with IOLService AOI which processes all IOL read and write requests.
// Status	Description
// 0	Operation completed successfully
// 	Status = 100 - 102, Ethernet IP MSG instruction errors - check communication parameters
// 100	IOL_SendMSG completed with error, check communication parameters
// 101	IOL_RecevieMSG completed with error, check communication parameters
// 110	IOL_Service Retry Limit exceeded
// 111	Slot specified not an IOLink master
// 	Status = 1000 to 1255, no response from device, connection error
// 1016	Device not connected or Port not configured as IOLink port
// 	Status = 2000 to 2255,  device response indicates error
// 2000	Device error, no details
// 2017	Device error, Index not available
// 2018	Device error, Subindex not available
// 2032	Device error, Service temporarily not available
// 2033	Device error, Service temporarily not available - local control
// 2034	Device error, Service temporarily not available - device control
// 2035	Device error, Index not writeable
// 2048	Device error, Parameter value out of range
// 2049	Device error, Parameter value above limit
// 2050	Device error, Parameter value below limit
// 2051	Device error, Parameter value length overrun (check IOLWrite precision/string length)
// 2052	Device error, Parameter value length underrun (check IOLWrite precision/string length)
// 2053	Device error, Function not available
// 2054	Device error, Function temporarily not available
// 2064	Device error, Parameter set invalid
// 2065	Device error, Inconsistent parameter set
// 2130	Device error, Application not ready
// 	Status = 3000 to 3255,   device response indicates vendor specific error
// 3000	Vendor specific error, no details
// 3001	Vendor specific error, vendor specific error number
// 3255	Vendor specific error, vendor specific error number
// 	Status = 7000 to 7255,  IOL-M Error Codes
// 7000	Unexpected write request instead of read request
// 7001	Decode error
// 7002	Port occupied by another task
// 	Status = 8000 to 8255,  IOL-M Error Codes
// 8000	Timeout when IOL-Ds or IOL-M ports are busy
// 8001	IOL Index out of range
// 8002	Port address greater than maximum
// 8003	Port function not supported
VAR_OUTPUT
   Done : BOOL; {access Read Only, visible}   // IOLRead completed successfully
   Error : BOOL; {access Read Only, visible}   // IOLRead completed with error, check status
   Pending : BOOL; {access Read Only, visible}   // IOLRead waiting to be processed
   Active : BOOL; {access Read Only, visible}   // IOLRead in progress
END_VAR
VAR_IN_OUT
   Common_Data : IOLRequest; {required}   // Shared IOL Data Area - must be identical on all requests
END_VAR
VAR_OUTPUT
   DoneCount : DINT; {access Read Only, visible}   // Number of operations completed successfully
   ErrorCount : DINT; {access Read Only, visible}   // Number of operations competed with error
   Status : INT; {access Read Only, visible}   // Status of last IOLRead
END_VAR
VAR_INPUT
   Read : BOOL;   // Rising edge triggers IOLink Read
   Read_Continuous : BOOL;   // Set to trigger IOLink Read repeatedly
   Slot : INT; {visible}   // IOLink Master slot number
   Port : INT; {visible}   // IOLink Master Port number, 1,2,3 or 4
   Index : INT; {visible}   // IOL Index number
   SubIndex : INT; {visible}   // IOL Subindex number
END_VAR
VAR_OUTPUT
   ReadData : DINT; {access Read Only, required}   // Data returned from IOLink device
END_VAR
VAR_INPUT
   R_8_Bit : BOOL;   // Indicates data received is 8 bit precision
   R_16_Bit : BOOL;   // Indicates data received is 16 bit precision
   R_32_Bit : BOOL;   // Indicates data received is 32 bit precision
   R_Sign_Extend : BOOL;   // Set to extend 8/16 bit precision data sign bit
   R_Swap_16 : BOOL;   // 16-bit AB->BA, 32-bit ABCD->BADC
   R_Swap_32 : BOOL;   // 32-bit ABCD->DCBA
   R_Swap_All : BOOL;   // 32-bit ABCD->CDBA
END_VAR
VAR
   MyHandle : INT;
   StartupDone : BOOL; {access None}
   Pending_or_Active : BOOL; {access None}
   Read_ONS : BOOL; {access None}
   StartupCount : DINT; {access None}
   ReadSignBit : DINT; {access None}
   ReadRequest : BOOL; {access None}
END_VAR

ROUTINE EnableInFalse   (* ladder *)
END_ROUTINE

ROUTINE Logic   (* ladder *)
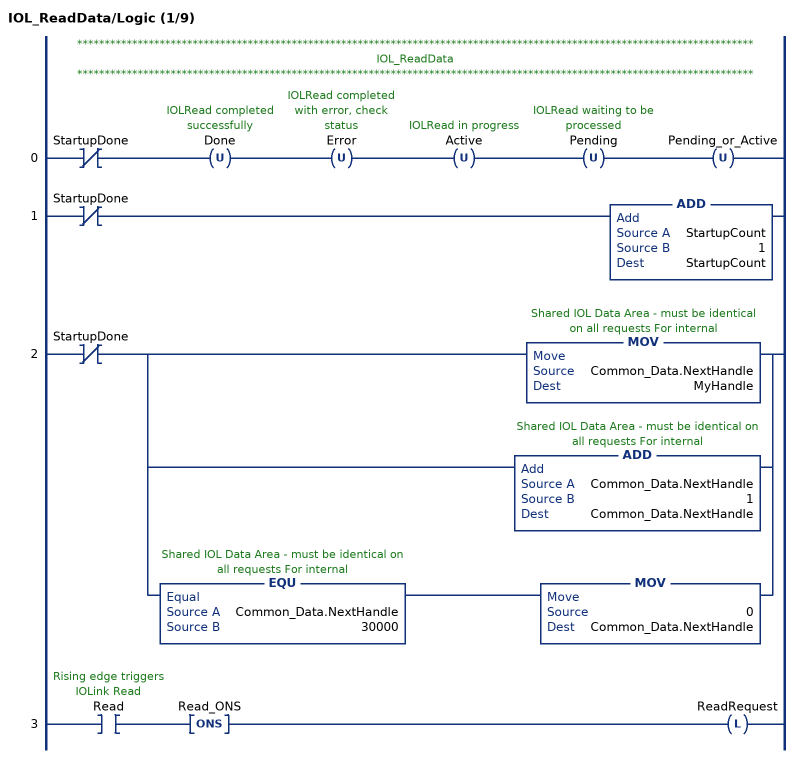
   // ***************************************************************************************************************************
   // IOL_ReadData
   // ***************************************************************************************************************************
   0: XIO(StartupDone)OTU(Done)OTU(Error)OTU(Active)OTU(Pending)OTU(Pending_or_Active);
   1: XIO(StartupDone)ADD(StartupCount,1,StartupCount);
   2: XIO(StartupDone)[MOV(Common_Data.NextHandle,MyHandle) ,ADD(Common_Data.NextHandle,1,Common_Data.NextHandle) ,EQU(Common_Data.NextHandle,30000) MOV(0,Common_Data.NextHandle) ];
   3: XIC(Read)ONS(Read_ONS)OTL(ReadRequest);
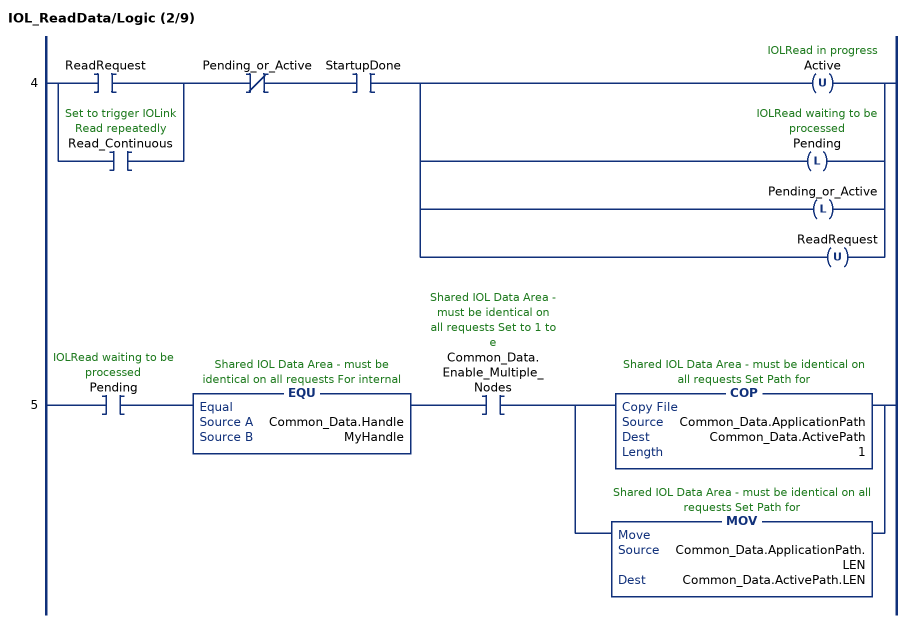
   4: [XIC(ReadRequest) ,XIC(Read_Continuous) ]XIO(Pending_or_Active)XIC(StartupDone)[OTU(Active) ,OTL(Pending) ,OTL(Pending_or_Active) ,OTU(ReadRequest) ];
   5: XIC(Pending)EQU(Common_Data.Handle,MyHandle)XIC(Common_Data.Enable_Multiple_Nodes)[COP(Common_Data.ApplicationPath,Common_Data.ActivePath,1) ,MOV(Common_Data.ApplicationPath.LEN,Common_Data.ActivePath.LEN) ];
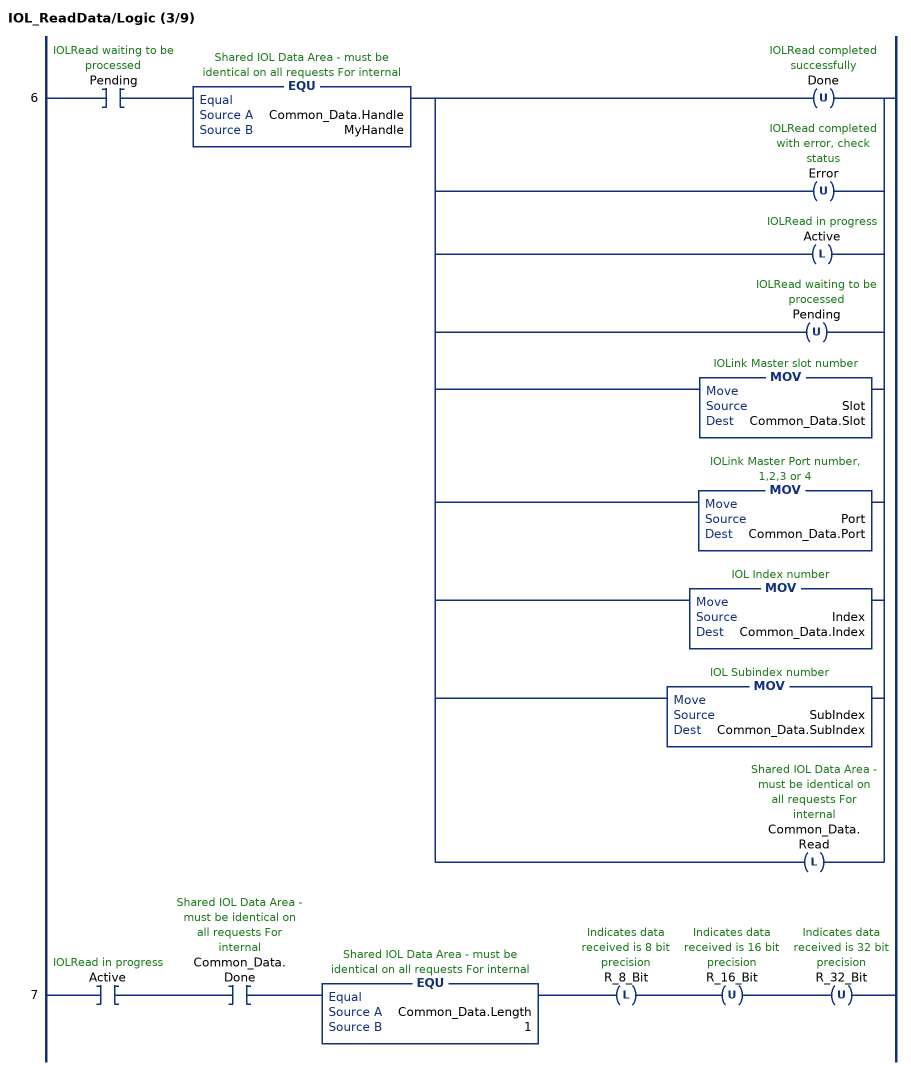
   6: XIC(Pending)EQU(Common_Data.Handle,MyHandle)[OTU(Done) ,OTU(Error) ,OTL(Active) ,OTU(Pending) ,MOV(Slot,Common_Data.Slot) ,MOV(Port,Common_Data.Port) ,MOV(Index,Common_Data.Index) ,MOV(SubIndex,Common_Data.SubIndex) ,OTL(Common_Data.Read) ];
   7: XIC(Active)XIC(Common_Data.Done)EQU(Common_Data.Length,1)OTL(R_8_Bit)OTU(R_16_Bit)OTU(R_32_Bit);
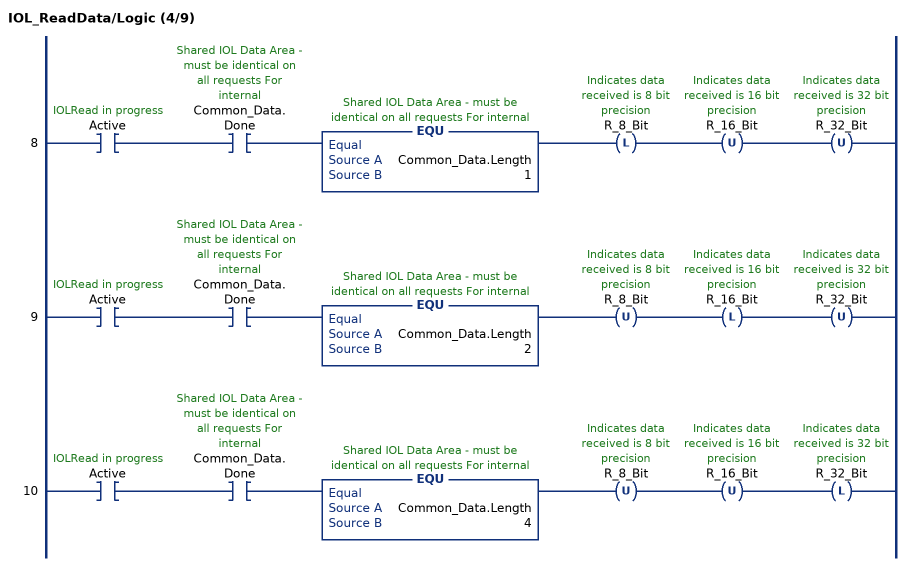
   8: XIC(Active)XIC(Common_Data.Done)EQU(Common_Data.Length,1)OTL(R_8_Bit)OTU(R_16_Bit)OTU(R_32_Bit);
   9: XIC(Active)XIC(Common_Data.Done)EQU(Common_Data.Length,2)OTU(R_8_Bit)OTL(R_16_Bit)OTU(R_32_Bit);
   10: XIC(Active)XIC(Common_Data.Done)EQU(Common_Data.Length,4)OTU(R_8_Bit)OTU(R_16_Bit)OTL(R_32_Bit);
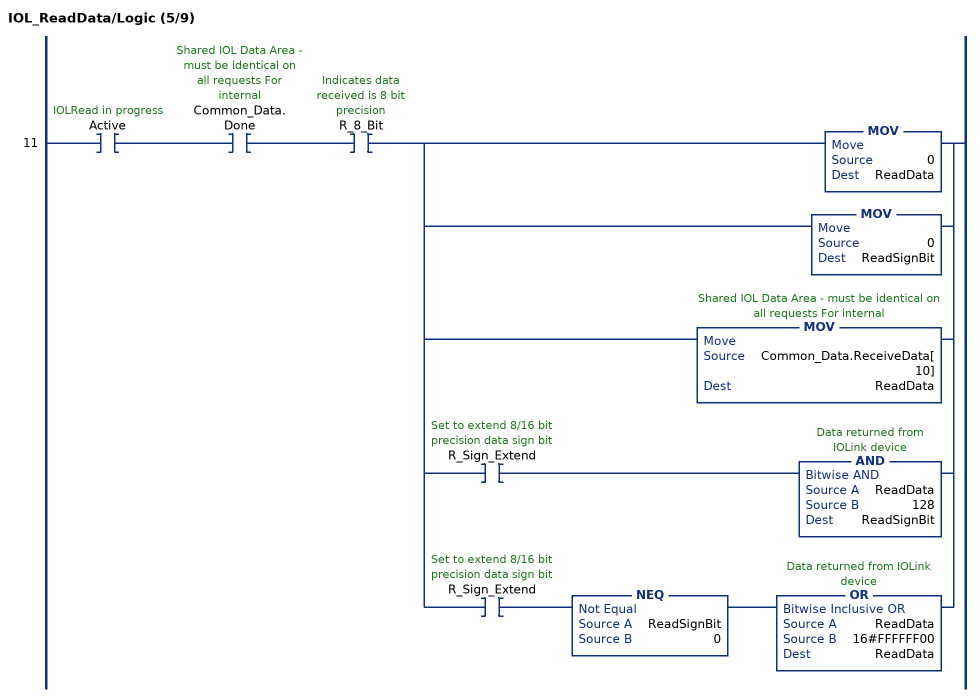
   11: XIC(Active)XIC(Common_Data.Done)XIC(R_8_Bit)[MOV(0,ReadData) ,MOV(0,ReadSignBit) ,MOV(Common_Data.ReceiveData[10],ReadData) ,XIC(R_Sign_Extend) AND(ReadData,128,ReadSignBit) ,XIC(R_Sign_Extend) NEQ(ReadSignBit,0) OR(ReadData,16#FFFFFF00,ReadData) ];
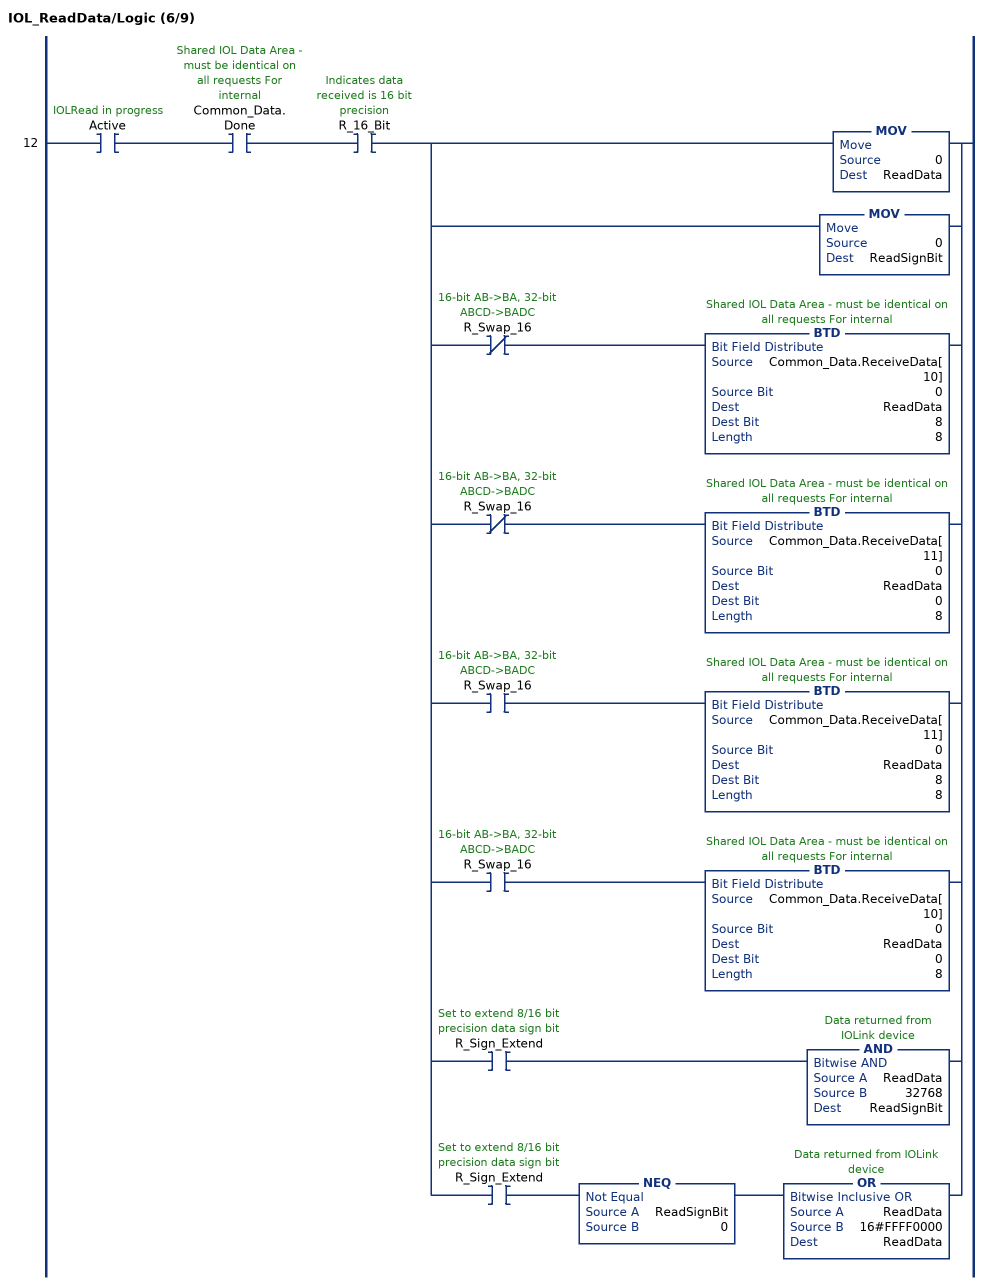
   12: XIC(Active)XIC(Common_Data.Done)XIC(R_16_Bit)[MOV(0,ReadData) ,MOV(0,ReadSignBit) ,XIO(R_Swap_16) BTD(Common_Data.ReceiveData[10],0,ReadData,8,8) ,XIO(R_Swap_16) BTD(Common_Data.ReceiveData[11],0,ReadData,0,8) ,XIC(R_Swap_16) BTD(Common_Data.ReceiveData[11],0,ReadData,8,8) ,XIC(R_Swap_16) BTD(Common_Data.ReceiveData[10],0,ReadData,0,8) ,XIC(R_Sign_Extend) AND(ReadData,32768,ReadSignBit) ,XIC(R_Sign_Extend) NEQ(ReadSignBit,0) OR(ReadData,16#FFFF0000,ReadData) ];
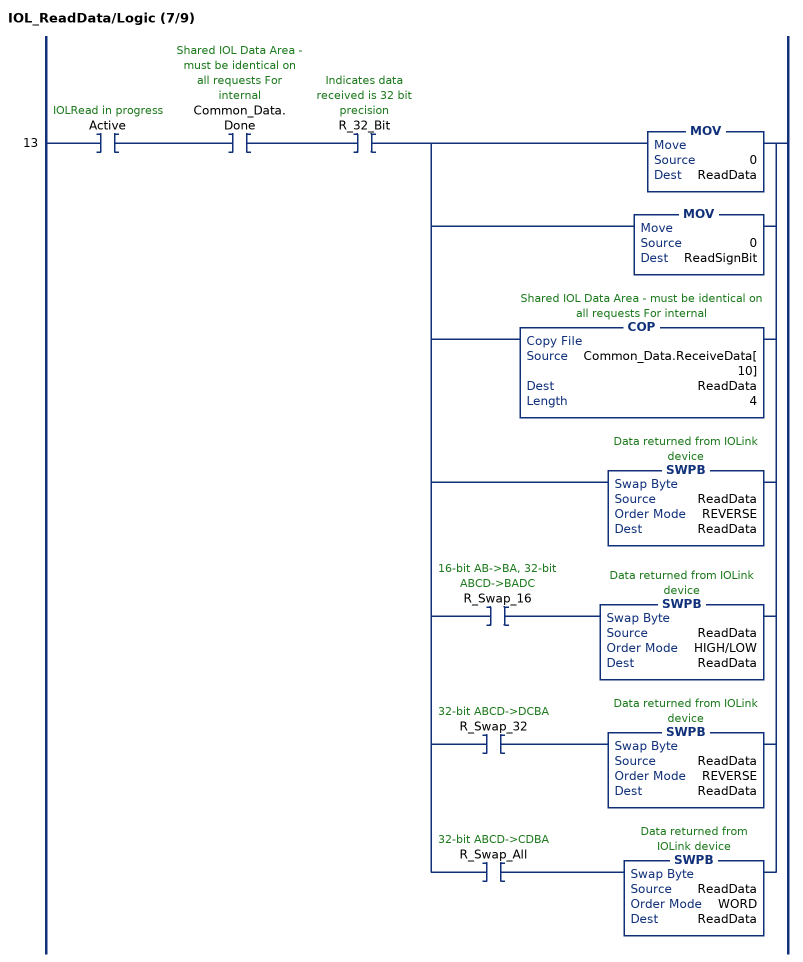
   13: XIC(Active)XIC(Common_Data.Done)XIC(R_32_Bit)[MOV(0,ReadData) ,MOV(0,ReadSignBit) ,COP(Common_Data.ReceiveData[10],ReadData,4) ,SWPB(ReadData,REVERSE,ReadData) ,XIC(R_Swap_16) SWPB(ReadData,HIGH/LOW,ReadData) ,XIC(R_Swap_32) SWPB(ReadData,REVERSE,ReadData) ,XIC(R_Swap_All) SWPB(ReadData,WORD,ReadData) ];
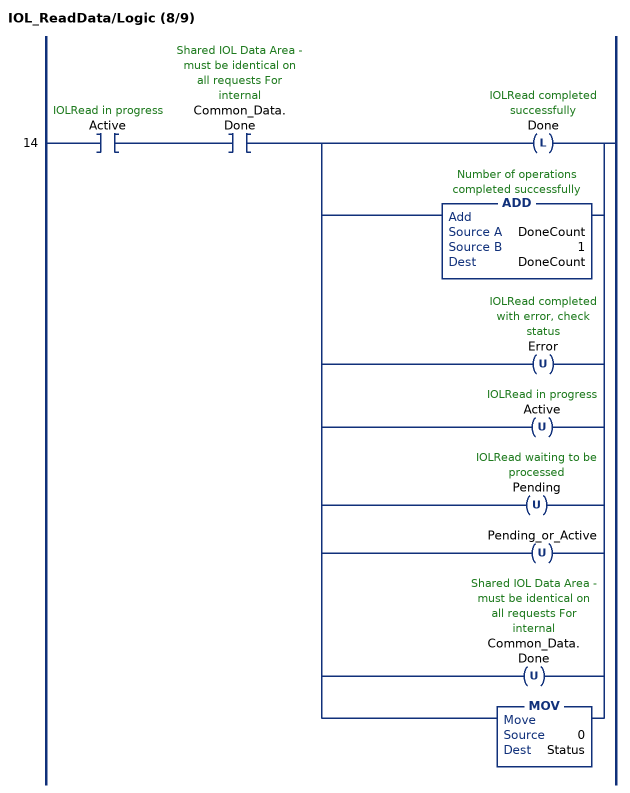
   14: XIC(Active)XIC(Common_Data.Done)[OTL(Done) ,ADD(DoneCount,1,DoneCount) ,OTU(Error) ,OTU(Active) ,OTU(Pending) ,OTU(Pending_or_Active) ,OTU(Common_Data.Done) ,MOV(0,Status) ];
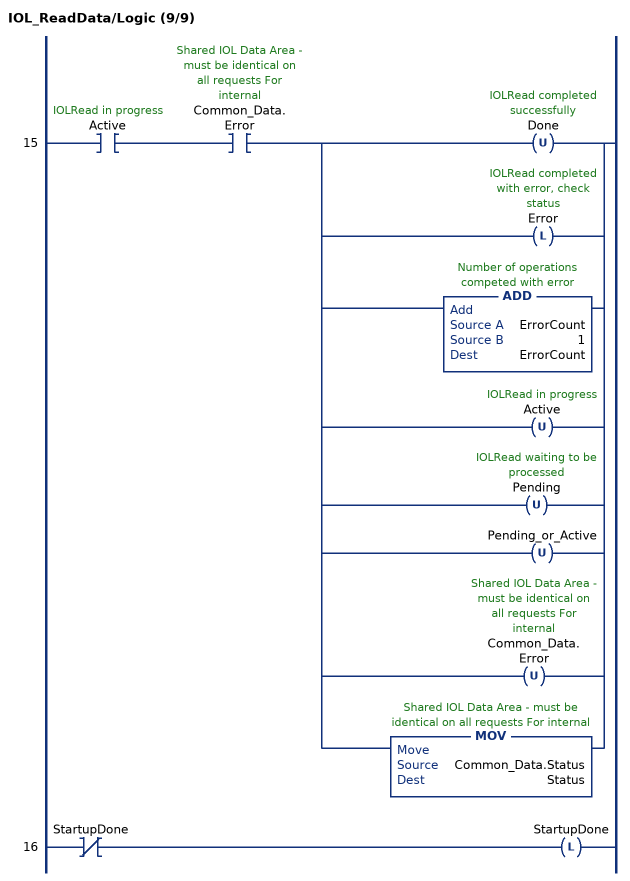
   15: XIC(Active)XIC(Common_Data.Error)[OTU(Done) ,OTL(Error) ,ADD(ErrorCount,1,ErrorCount) ,OTU(Active) ,OTU(Pending) ,OTU(Pending_or_Active) ,OTU(Common_Data.Error) ,MOV(Common_Data.Status,Status) ];
   16: XIO(StartupDone)OTL(StartupDone);
END_ROUTINE
